KUKA KRL program: MyProgram_211().src

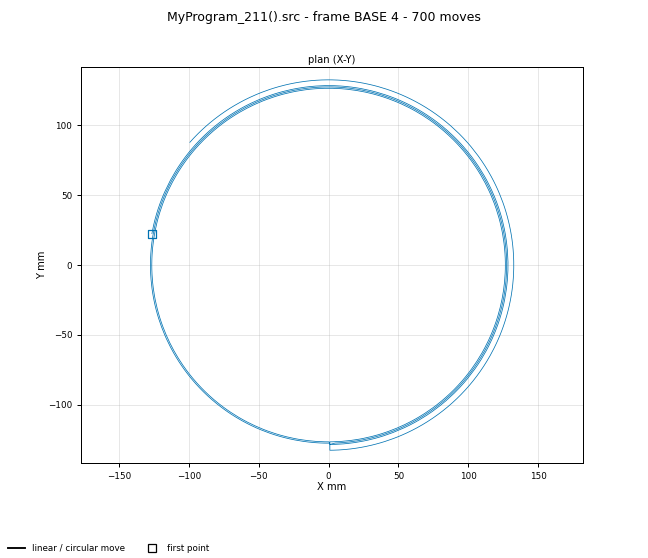
[picture p0: tool path of MyProgram_211().src in frame BASE 4, 700 of 700 moves have a stored position in this frame; points joined in program order, loops and branches not executed]
&ACCESS RVP
&REL 1
&PARAM TEMPLATE = C:\KRC\Roboter\Template\vorgabe
&PARAM EDITMASK = *
DEF MyProgram_211()
; ---- Setting reference (Base) ----
$BASE = BASE_DATA[4]

; --------------------------
; ---- Setting tool (TCP) ----
$TOOL = TOOL_DATA[3]
; --------------------------

$VEL.CP = VEL_APROX_PRINT
Startdeposition()
$VEL.CP = VEL_PRINT
LIN {X -126.5024,Y 22.5306,Z 149,A 167.0251,B 21.3355,C -0.911,E1 21.1965,E2 280.5276} C_DIS
LIN {X -125.8833,Y 25.7659,Z 149,A 165.5743,B 21.3353,C -0.9164,E1 21.1973,E2 281.9739} C_DIS
LIN {X -125.2551,Y 28.6636,Z 149,A 164.2083,B 21.3353,C -0.9188,E1 21.1981,E2 283.3427} C_DIS
LIN {X -124.3308,Y 32.4464,Z 149,A 161.9232,B 21.3358,C -0.9032,E1 21.1998,E2 285.6871} C_DIS
LIN {X -123.1759,Y 36.584,Z 149,A 160.1986,B 21.3353,C -0.9164,E1 21.2011,E2 287.387} C_DIS
LIN {X -122.1569,Y 39.8588,Z 149,A 159.0156,B 21.3346,C -0.9344,E1 21.2021,E2 288.5283} C_DIS
LIN {X -120.7931,Y 43.8121,Z 149,A 156.8151,B 21.3349,C -0.9272,E1 21.2042,E2 290.7636} C_DIS
LIN {X -118.9565,Y 48.5809,Z 149,A 154.7384,B 21.3342,C -0.9418,E1 21.2063,E2 292.8137} C_DIS
LIN {X -117.417,Y 52.1895,Z 149,A 152.9389,B 21.3342,C -0.9451,E1 21.2083,E2 294.616} C_DIS
LIN {X -113.3111,Y 60.5932,Z 149,A 148.9309,B 21.3333,C -0.9635,E1 21.2133,E2 298.5988} C_DIS
LIN {X -109.5371,Y 67.1752,Z 149,A 145.6179,B 21.3328,C -0.9757,E1 21.2179,E2 301.8985} C_DIS
LIN {X -107.9534,Y 69.6925,Z 149,A 143.9828,B 21.3332,C -0.9674,E1 21.2204,E2 303.5666} C_DIS
LIN {X -105.4695,Y 73.3966,Z 149,A 141.5266,B 21.3337,C -0.9547,E1 21.2243,E2 306.0723} C_DIS
LIN {X -102.7831,Y 77.1145,Z 149,A 139.5857,B 21.3333,C -0.9642,E1 21.2275,E2 307.9982} C_DIS
LIN {X -100.3563,Y 80.247,Z 149,A 138.1638,B 21.3325,C -0.9821,E1 21.2299,E2 309.3785} C_DIS
LIN {X -97.498,Y 83.6963,Z 149,A 136.0509,B 21.3325,C -0.9827,E1 21.2338,E2 311.5014} C_DIS
LIN {X -95.072,Y 86.442,Z 149,A 134.5353,B 21.3321,C -0.9913,E1 21.2366,E2 313.0012} C_DIS
LIN {X -92.0357,Y 89.6687,Z 149,A 132.5092,B 21.332,C -0.9941,E1 21.2405,E2 315.0301} C_DIS
LIN {X -88.8889,Y 92.7883,Z 149,A 130.6084,B 21.3316,C -1.0016,E1 21.2443,E2 316.9194} C_DIS
LIN {X -86.2647,Y 95.2328,Z 149,A 129.1349,B 21.3313,C -1.0102,E1 21.2472,E2 318.3764} C_DIS
LIN {X -83.3834,Y 97.7657,Z 149,A 127.3435,B 21.3313,C -1.0108,E1 21.251,E2 320.1746} C_DIS
LIN {X -80.3668,Y 100.2607,Z 149,A 125.424,B 21.3313,C -1.0077,E1 21.2552,E2 322.1114} C_DIS
LIN {X -76.5633,Y 103.194,Z 149,A 123.3887,B 21.331,C -1.0163,E1 21.2597,E2 324.1317} C_DIS
LIN {X -73.2443,Y 105.5755,Z 149,A 121.5811,B 21.3308,C -1.0204,E1 21.2638,E2 325.9353} C_DIS
LIN {X -70.1708,Y 107.6429,Z 149,A 119.8567,B 21.3308,C -1.0206,E1 21.2679,E2 327.6658} C_DIS
LIN {X -66.1096,Y 110.1838,Z 149,A 117.7568,B 21.3305,C -1.0259,E1 21.2728,E2 329.759} C_DIS
LIN {X -62.338,Y 112.3601,Z 149,A 115.4206,B 21.3311,C -1.0136,E1 21.2786,E2 332.1374} C_DIS
LIN {X -59.0857,Y 114.1043,Z 149,A 114.1862,B 21.3302,C -1.0326,E1 21.2816,E2 333.3234} C_DIS
LIN {X -55.8111,Y 115.7399,Z 149,A 112.3225,B 21.3305,C -1.0258,E1 21.2863,E2 335.2114} C_DIS
LIN {X -50.8834,Y 117.9885,Z 149,A 110.1116,B 21.33,C -1.0375,E1 21.2919,E2 337.3965} C_DIS
LIN {X -47.6091,Y 119.3482,Z 149,A 108.3813,B 21.3302,C -1.0336,E1 21.2964,E2 339.1421} C_DIS
LIN {X -43.4647,Y 120.9184,Z 149,A 105.8791,B 21.331,C -1.015,E1 21.3031,E2 341.7016} C_DIS
LIN {X -38.7505,Y 122.5111,Z 149,A 104.4896,B 21.3294,C -1.0509,E1 21.3065,E2 342.9952} C_DIS
LIN {X -36.1903,Y 123.2911,Z 149,A 103.0975,B 21.3297,C -1.0441,E1 21.3103,E2 344.4089} C_DIS
LIN {X -32.8603,Y 124.2204,Z 149,A 101.6079,B 21.3295,C -1.0477,E1 21.3143,E2 345.8911} C_DIS
LIN {X -29.7621,Y 124.9992,Z 149,A 100.1887,B 21.3295,C -1.0493,E1 21.3181,E2 347.3085} C_DIS
LIN {X -26.6465,Y 125.7006,Z 149,A 98.734,B 21.3295,C -1.0492,E1 21.3221,E2 348.7656} C_DIS
LIN {X -22.5065,Y 126.5067,Z 149,A 96.5684,B 21.3299,C -1.039,E1 21.3282,E2 350.9621} C_DIS
LIN {X -17.6004,Y 127.2833,Z 149,A 94.5907,B 21.3294,C -1.05,E1 21.3335,E2 352.9113} C_DIS
LIN {X -13.9215,Y 127.7369,Z 149,A 92.2906,B 21.3306,C -1.0244,E1 21.3401,E2 355.2835} C_DIS
LIN {X -8.9034,Y 128.1852,Z 149,A 90.7884,B 21.3292,C -1.0558,E1 21.3441,E2 356.7} C_DIS
LIN {X -2.7081,Y 128.466,Z 149,A 88.0474,B 21.3291,C -1.0576,E1 21.3517,E2 359.4369} C_DIS
LIN {X 4.2169,Y 128.4248,Z 149,A 84.9282,B 21.3291,C -1.0567,E1 21.3604,E2 362.5581} C_DIS
LIN {X 8.7162,Y 128.1989,Z 149,A 82.8985,B 21.3291,C -1.0558,E1 21.3661,E2 364.5895} C_DIS
LIN {X 12.1904,Y 127.9137,Z 149,A 80.8062,B 21.3302,C -1.0331,E1 21.3721,E2 366.7424} C_DIS
LIN {X 16.289,Y 127.4571,Z 149,A 79.4266,B 21.3293,C -1.0519,E1 21.3757,E2 368.0693} C_DIS
LIN {X 20.9637,Y 126.7716,Z 149,A 77.6065,B 21.3288,C -1.0633,E1 21.3807,E2 369.856} C_DIS
LIN {X 23.6917,Y 126.2908,Z 149,A 76.0677,B 21.3294,C -1.05,E1 21.385,E2 371.4294} C_DIS
LIN {X 27.1575,Y 125.5903,Z 149,A 74.566,B 21.3294,C -1.0524,E1 21.3891,E2 372.9223} C_DIS
LIN {X 30.1689,Y 124.9011,Z 149,A 73.1257,B 21.3294,C -1.0489,E1 21.393,E2 374.3696} C_DIS
LIN {X 33.9154,Y 123.9383,Z 149,A 71.31,B 21.3297,C -1.0439,E1 21.3979,E2 376.1957} C_DIS
LIN {X 37.8426,Y 122.7942,Z 149,A 69.6544,B 21.3294,C -1.0497,E1 21.4023,E2 377.8318} C_DIS
LIN {X 40.6135,Y 121.9055,Z 149,A 68.3282,B 21.3295,C -1.0474,E1 21.4058,E2 379.1614} C_DIS
LIN {X 43.7376,Y 120.82,Z 149,A 66.4377,B 21.3304,C -1.0283,E1 21.4109,E2 381.0995} C_DIS
LIN {X 47.3652,Y 119.4465,Z 149,A 64.6738,B 21.3306,C -1.0251,E1 21.4155,E2 382.8676} C_DIS
LIN {X 50.8844,Y 117.9881,Z 149,A 63.4384,B 21.3298,C -1.0431,E1 21.4186,E2 384.0502} C_DIS
LIN {X 54.0438,Y 116.5747,Z 149,A 61.8787,B 21.3298,C -1.0406,E1 21.4225,E2 385.6122} C_DIS
LIN {X 57.0953,Y 115.1112,Z 149,A 60.3886,B 21.3299,C -1.0395,E1 21.4263,E2 387.1004} C_DIS
LIN {X 59.9976,Y 113.6255,Z 149,A 58.904,B 21.3301,C -1.0362,E1 21.43,E2 388.589} C_DIS
LIN {X 63.8911,Y 111.4849,Z 149,A 56.7721,B 21.3305,C -1.0269,E1 21.4352,E2 390.7389} C_DIS
LIN {X 66.7791,Y 109.7796,Z 149,A 55.4128,B 21.3303,C -1.0305,E1 21.4384,E2 392.0832} C_DIS
LIN {X 70.0603,Y 107.7147,Z 149,A 53.6927,B 21.3304,C -1.0282,E1 21.4425,E2 393.8031} C_DIS
LIN {X 74.7579,Y 104.509,Z 149,A 51.1929,B 21.3306,C -1.0255,E1 21.4482,E2 396.3} C_DIS
LIN {X 77.9903,Y 102.1195,Z 149,A 49.3589,B 21.3308,C -1.0205,E1 21.4523,E2 398.1398} C_DIS
LIN {X 81.4914,Y 99.3483,Z 149,A 47.3921,B 21.3309,C -1.0179,E1 21.4566,E2 400.1051} C_DIS
LIN {X 84.7295,Y 96.6018,Z 149,A 45.5153,B 21.331,C -1.0149,E1 21.4605,E2 401.9811} C_DIS
LIN {X 88.9751,Y 92.7059,Z 149,A 42.9302,B 21.3313,C -1.009,E1 21.4658,E2 404.57} C_DIS
LIN {X 91.0131,Y 90.7057,Z 149,A 41.2496,B 21.3322,C -0.9883,E1 21.4693,E2 406.2985} C_DIS
LIN {X 93.9321,Y 87.6793,Z 149,A 39.8186,B 21.3316,C -1.0037,E1 21.4719,E2 407.6799} C_DIS
LIN {X 96.6382,Y 84.6877,Z 149,A 37.9954,B 21.3318,C -0.9986,E1 21.4753,E2 409.5075} C_DIS
LIN {X 99.4168,Y 81.4076,Z 149,A 36.0873,B 21.332,C -0.9945,E1 21.4787,E2 411.4164} C_DIS
LIN {X 102.2616,Y 77.8046,Z 149,A 34.0421,B 21.3322,C -0.9896,E1 21.4822,E2 413.4633} C_DIS
LIN {X 104.8267,Y 74.3124,Z 149,A 31.6772,B 21.3332,C -0.9656,E1 21.4861,E2 415.8801} C_DIS
LIN {X 107.3529,Y 70.6132,Z 149,A 30.6055,B 21.3316,C -1.0018,E1 21.4877,E2 416.8465} C_DIS
LIN {X 111.3736,Y 64.0852,Z 149,A 26.928,B 21.3326,C -0.9812,E1 21.4931,E2 420.5581} C_DIS
LIN {X 113.0317,Y 61.1133,Z 149,A 25.2168,B 21.3331,C -0.9684,E1 21.4954,E2 422.2937} C_DIS
LIN {X 115.1112,Y 57.0953,Z 149,A 23.2364,B 21.3333,C -0.9645,E1 21.4979,E2 424.2721} C_DIS
LIN {X 116.7392,Y 53.6882,Z 149,A 21.636,B 21.3333,C -0.9635,E1 21.4998,E2 425.8648} C_DIS
LIN {X 118.8712,Y 48.7873,Z 149,A 19.1595,B 21.3338,C -0.9525,E1 21.5025,E2 428.3552} C_DIS
LIN {X 120.5097,Y 44.5879,Z 149,A 17.2936,B 21.3338,C -0.9532,E1 21.5043,E2 430.207} C_DIS
LIN {X 121.7655,Y 41.0342,Z 149,A 15.5898,B 21.334,C -0.9472,E1 21.5059,E2 431.9158} C_DIS
LIN {X 122.8444,Y 37.6788,Z 149,A 14.0311,B 21.3342,C -0.9431,E1 21.5072,E2 433.4751} C_DIS
LIN {X 123.7755,Y 34.4973,Z 149,A 12.6305,B 21.3342,C -0.9421,E1 21.5083,E2 434.8687} C_DIS
LIN {X 124.6792,Y 31.0778,Z 149,A 11.0066,B 21.3345,C -0.9352,E1 21.5094,E2 436.5003} C_DIS
LIN {X 125.8354,Y 26.0013,Z 149,A 8.9227,B 21.3344,C -0.9389,E1 21.5107,E2 438.5598} C_DIS
LIN {X 126.5495,Y 22.2671,Z 149,A 7.0765,B 21.3349,C -0.9268,E1 21.5116,E2 440.4261} C_DIS
LIN {X 127.4203,Y 16.5703,Z 149,A 4.5861,B 21.3351,C -0.9224,E1 21.5126,E2 442.9112} C_DIS
LIN {X 128.0462,Y 10.709,Z 149,A 1.804,B 21.3357,C -0.9071,E1 21.5134,E2 445.7154} C_DIS
LIN {X 128.4745,Y 2.2,Z 149,A -2.7502,B 21.3375,C -0.8609,E1 21.5138,E2 450.3633} C_DIS
LIN {X 128.4331,Y -3.9504,Z 149,A -5.6329,B 21.3381,C -0.8459,E1 21.5136,E2 453.2665} C_DIS
LIN {X 128.0339,Y -10.8549,Z 149,A -7.5384,B 21.3364,C -0.8894,E1 21.5132,E2 455.0399} C_DIS
LIN {X 127.3738,Y -16.9253,Z 149,A -10.2869,B 21.3368,C -0.8795,E1 21.5124,E2 457.796} C_DIS
LIN {X 126.0458,Y -24.9673,Z 149,A -14.0539,B 21.3375,C -0.8619,E1 21.5106,E2 461.5848} C_DIS
LIN {X 125.281,Y -28.5505,Z 149,A -15.5989,B 21.3375,C -0.8608,E1 21.5096,E2 463.122} C_DIS
LIN {X 124.5398,Y -31.6271,Z 149,A -16.9744,B 21.3376,C -0.858,E1 21.5087,E2 464.4957} C_DIS
LIN {X 123.6426,Y -34.9726,Z 149,A -18.5415,B 21.3378,C -0.8521,E1 21.5075,E2 466.0681} C_DIS
LIN {X 122.3986,Y -39.1026,Z 149,A -20.4262,B 21.338,C -0.848,E1 21.506,E2 467.9514} C_DIS
LIN {X 121.3036,Y -42.3787,Z 149,A -21.9571,B 21.3382,C -0.8436,E1 21.5046,E2 469.4838} C_DIS
LIN {X 119.49,Y -47.2557,Z 149,A -24.2295,B 21.3383,C -0.8387,E1 21.5024,E2 471.7545} C_DIS
LIN {X 118.2879,Y -50.1888,Z 149,A -25.632,B 21.3385,C -0.835,E1 21.5009,E2 473.1581} C_DIS
LIN {X 117.1157,Y -52.863,Z 149,A -26.9554,B 21.3387,C -0.8301,E1 21.4994,E2 474.4861} C_DIS
LIN {X 114.5241,Y -58.2632,Z 149,A -29.6054,B 21.3389,C -0.8232,E1 21.4961,E2 477.1381} C_DIS
LIN {X 112.8123,Y -61.5165,Z 149,A -31.3116,B 21.3392,C -0.8154,E1 21.4938,E2 478.8549} C_DIS
LIN {X 109.4302,Y -67.3494,Z 149,A -33.9605,B 21.3389,C -0.8231,E1 21.4902,E2 481.4666} C_DIS
LIN {X 107.0779,Y -71.0307,Z 149,A -36.2183,B 21.3396,C -0.8036,E1 21.4867,E2 483.7642} C_DIS
LIN {X 104.7211,Y -74.4612,Z 149,A -38.0778,B 21.3398,C -0.7984,E1 21.4837,E2 485.6271} C_DIS
LIN {X 99.2501,Y -81.6115,Z 149,A -41.8391,B 21.3398,C -0.7992,E1 21.4773,E2 489.3649} C_DIS
LIN {X 97.2041,Y -84.0375,Z 149,A -44.077,B 21.3412,C -0.7586,E1 21.4731,E2 491.7015} C_DIS
LIN {X 93.7509,Y -87.8736,Z 149,A -46.4121,B 21.3414,C -0.7515,E1 21.4686,E2 494.0441} C_DIS
LIN {X 90,Y -91.7109,Z 149,A -48.0087,B 21.3404,C -0.7814,E1 21.4656,E2 495.551} C_DIS
LIN {X 84.0776,Y -97.1696,Z 149,A -51.4099,B 21.3404,C -0.7816,E1 21.4587,E2 498.9351} C_DIS
LIN {X 80.033,Y -100.5266,Z 149,A -53.9677,B 21.3409,C -0.7669,E1 21.4531,E2 501.5215} C_DIS
LIN {X 74.3559,Y -104.7959,Z 149,A -57.3669,B 21.3415,C -0.7501,E1 21.4454,E2 504.9523} C_DIS
LIN {X 70.2672,Y -107.5803,Z 149,A -59.4392,B 21.3415,C -0.7517,E1 21.4406,E2 507.0118} C_DIS
LIN {X 64.9358,Y -110.879,Z 149,A -62.1325,B 21.3415,C -0.7511,E1 21.4342,E2 509.6966} C_DIS
LIN {X 61.8538,Y -112.6283,Z 149,A -63.6817,B 21.3415,C -0.7498,E1 21.4304,E2 511.2441} C_DIS
LIN {X 57.9866,Y -114.665,Z 149,A -65.6063,B 21.3415,C -0.7477,E1 21.4256,E2 513.168} C_DIS
LIN {X 54.2584,Y -116.4755,Z 149,A -67.4216,B 21.3416,C -0.7463,E1 21.421,E2 514.9816} C_DIS
LIN {X 46.0167,Y -119.9717,Z 149,A -71.304,B 21.3416,C -0.7454,E1 21.4111,E2 518.8555} C_DIS
LIN {X 39.0159,Y -122.4263,Z 149,A -74.6753,B 21.3419,C -0.7385,E1 21.4022,E2 522.2378} C_DIS
LIN {X 35.9952,Y -123.3483,Z 149,A -76.0894,B 21.3419,C -0.7367,E1 21.3983,E2 523.6538} C_DIS
LIN {X 32.7815,Y -124.2414,Z 149,A -77.6265,B 21.3421,C -0.733,E1 21.3942,E2 525.1981} C_DIS
LIN {X 28.0427,Y -125.397,Z 149,A -79.7469,B 21.3421,C -0.7333,E1 21.3884,E2 527.3141} C_DIS
LIN {X 25.0664,Y -126.0256,Z 149,A -81.2666,B 21.3423,C -0.7251,E1 21.3842,E2 528.8541} C_DIS
LIN {X 18.7391,Y -127.1205,Z 149,A -83.9386,B 21.3421,C -0.7313,E1 21.3769,E2 531.5058} C_DIS
LIN {X 13.5131,Y -127.7809,Z 149,A -86.3427,B 21.3422,C -0.7275,E1 21.3702,E2 533.918} C_DIS
LIN {X 10.7784,Y -128.0404,Z 149,A -88.4747,B 21.3435,C -0.6883,E1 21.364,E2 536.1563} C_DIS
LIN {X 4.483,Y -128.4161,Z 149,A -90.14,B 21.342,C -0.7361,E1 21.3597,E2 537.6897} C_DIS
LIN {X 0.927,Y -128.4536,Z 149,A -91.6085,B 21.3418,C -0.7412,E1 21.3557,E2 539.144} C_DIS
Enddeposition()
LIN {X 0.927,Y -128.4536,Z 149,A -91.6085,B 21.3418,C -0.7412,E1 21.3557,E2 539.144} C_DIS
Startdeposition()
$VEL.CP = VEL_PRINT
LIN {X 4.7464,Y -127.4561,Z 149,A -89.2402,B 20.1151,C -0.5881,E1 20.1307,E2 537.0751} C_DIS
LIN {X 10.6568,Y -127.0982,Z 149,A -86.5313,B 20.1151,C -0.5911,E1 20.1383,E2 534.3589} C_DIS
LIN {X 14.5444,Y -126.7134,Z 149,A -84.6534,B 20.1148,C -0.5971,E1 20.1435,E2 532.4654} C_DIS
LIN {X 20.2771,Y -125.9232,Z 149,A -81.9669,B 20.1147,C -0.6023,E1 20.151,E2 529.7668} C_DIS
LIN {X 24.4978,Y -125.1705,Z 149,A -80.3198,B 20.115,C -0.5923,E1 20.1554,E2 528.1511} C_DIS
LIN {X 27.9449,Y -124.4458,Z 149,A -78.843,B 20.115,C -0.5894,E1 20.1594,E2 526.6854} C_DIS
LIN {X 30.1986,Y -123.9177,Z 149,A -77.5315,B 20.1147,C -0.6015,E1 20.1631,E2 525.3411} C_DIS
LIN {X 34.1976,Y -122.8739,Z 149,A -75.854,B 20.1149,C -0.596,E1 20.1675,E2 523.6831} C_DIS
LIN {X 36.6862,Y -122.1557,Z 149,A -74.6923,B 20.1149,C -0.5971,E1 20.1706,E2 522.5205} C_DIS
LIN {X 39.4672,Y -121.2858,Z 149,A -73.0131,B 20.1144,C -0.614,E1 20.1752,E2 520.7964} C_DIS
LIN {X 42.6116,Y -120.2171,Z 149,A -71.9127,B 20.1148,C -0.5995,E1 20.178,E2 519.7408} C_DIS
LIN {X 45.5503,Y -119.1348,Z 149,A -70.4147,B 20.1146,C -0.6051,E1 20.1819,E2 518.2307} C_DIS
LIN {X 48.5804,Y -117.9311,Z 149,A -69.0819,B 20.1147,C -0.6017,E1 20.1854,E2 516.9118} C_DIS
LIN {X 52.8709,Y -116.0715,Z 149,A -66.7448,B 20.1143,C -0.6145,E1 20.1914,E2 514.5447} C_DIS
LIN {X 56.4413,Y -114.3756,Z 149,A -65.1143,B 20.1144,C -0.6112,E1 20.1955,E2 512.9292} C_DIS
LIN {X 59.6772,Y -112.7218,Z 149,A -63.326,B 20.1142,C -0.6204,E1 20.1999,E2 511.1208} C_DIS
LIN {X 62.6986,Y -111.0713,Z 149,A -61.2287,B 20.1134,C -0.6464,E1 20.2052,E2 508.9562} C_DIS
LIN {X 67.3098,Y -108.3387,Z 149,A -59.4808,B 20.1141,C -0.6227,E1 20.2092,E2 507.2838} C_DIS
LIN {X 71.0985,Y -105.8914,Z 149,A -57.6121,B 20.1141,C -0.6199,E1 20.2135,E2 505.4312} C_DIS
LIN {X 73.1065,Y -104.5152,Z 149,A -56.4889,B 20.1141,C -0.6233,E1 20.2161,E2 504.3031} C_DIS
LIN {X 76.7611,Y -101.8608,Z 149,A -54.3562,B 20.1138,C -0.6317,E1 20.2209,E2 502.1555} C_DIS
LIN {X 80.2186,Y -99.161,Z 149,A -52.4189,B 20.1138,C -0.6345,E1 20.2251,E2 500.2196} C_DIS
LIN {X 82.5731,Y -97.2089,Z 149,A -50.8736,B 20.1134,C -0.6448,E1 20.2285,E2 498.6521} C_DIS
LIN {X 87.5263,Y -92.7741,Z 149,A -48.1006,B 20.1135,C -0.6424,E1 20.2342,E2 495.9003} C_DIS
LIN {X 90.4671,Y -89.9088,Z 149,A -46.473,B 20.1137,C -0.6374,E1 20.2374,E2 494.2957} C_DIS
LIN {X 93.8115,Y -86.4135,Z 149,A -43.914,B 20.113,C -0.6592,E1 20.2424,E2 491.6879} C_DIS
LIN {X 97.1984,Y -82.5855,Z 149,A -41.8392,B 20.1131,C -0.6554,E1 20.2461,E2 489.636} C_DIS
LIN {X 99.9768,Y -79.1998,Z 149,A -39.5317,B 20.1125,C -0.6751,E1 20.2502,E2 487.2853} C_DIS
LIN {X 102.1851,Y -76.3291,Z 149,A -38.3444,B 20.113,C -0.6604,E1 20.2521,E2 486.1475} C_DIS
LIN {X 104.4711,Y -73.1699,Z 149,A -36.4435,B 20.1126,C -0.6715,E1 20.2552,E2 484.2264} C_DIS
LIN {X 106.6586,Y -69.9421,Z 149,A -34.6369,B 20.1124,C -0.6787,E1 20.258,E2 482.4106} C_DIS
LIN {X 109.2731,Y -65.7825,Z 149,A -32.7045,B 20.1126,C -0.6729,E1 20.2608,E2 480.5073} C_DIS
LIN {X 111.4856,Y -61.9588,Z 149,A -30.5627,B 20.1122,C -0.6853,E1 20.2638,E2 478.3437} C_DIS
LIN {X 113.45,Y -58.2812,Z 149,A -28.6777,B 20.112,C -0.6912,E1 20.2663,E2 476.4543} C_DIS
LIN {X 115.32,Y -54.4884,Z 149,A -26.8032,B 20.1118,C -0.6957,E1 20.2685,E2 474.5798} C_DIS
LIN {X 116.9069,Y -50.9937,Z 149,A -25.1424,B 20.1118,C -0.698,E1 20.2704,E2 472.9237} C_DIS
LIN {X 118.0942,Y -48.1815,Z 149,A -23.7507,B 20.1116,C -0.703,E1 20.2719,E2 471.5275} C_DIS
LIN {X 119.5931,Y -44.3294,Z 149,A -21.8766,B 20.1114,C -0.7093,E1 20.2738,E2 469.6483} C_DIS
LIN {X 120.9543,Y -40.4662,Z 149,A -20.1202,B 20.1113,C -0.7113,E1 20.2753,E2 467.8988} C_DIS
LIN {X 122.2021,Y -36.5323,Z 149,A -18.2143,B 20.111,C -0.7192,E1 20.2769,E2 465.984} C_DIS
LIN {X 123.1596,Y -33.155,Z 149,A -16.9029,B 20.1112,C -0.7125,E1 20.2779,E2 464.7012} C_DIS
LIN {X 123.8345,Y -30.544,Z 149,A -15.6412,B 20.111,C -0.7184,E1 20.2787,E2 463.4318} C_DIS
LIN {X 124.6724,Y -26.9119,Z 149,A -13.9981,B 20.111,C -0.7223,E1 20.2797,E2 461.7896} C_DIS
LIN {X 125.4148,Y -23.2198,Z 149,A -11.8715,B 20.1101,C -0.7464,E1 20.2809,E2 459.6092} C_DIS
LIN {X 125.9857,Y -19.8801,Z 149,A -10.6929,B 20.1104,C -0.7363,E1 20.2814,E2 458.4687} C_DIS
LIN {X 126.4932,Y -16.3412,Z 149,A -9.1436,B 20.1104,C -0.7389,E1 20.282,E2 456.9234} C_DIS
LIN {X 127.0258,Y -11.508,Z 149,A -6.8324,B 20.1099,C -0.7512,E1 20.2826,E2 454.594} C_DIS
LIN {X 127.4544,Y -4.79,Z 149,A -3.9482,B 20.1098,C -0.7547,E1 20.2831,E2 451.7216} C_DIS
LIN {X 127.5431,Y -0.7829,Z 149,A -2.3585,B 20.1098,C -0.7512,E1 20.2831,E2 450.1539} C_DIS
LIN {X 127.5386,Y 1.3934,Z 149,A -1.0105,B 20.1092,C -0.7703,E1 20.2831,E2 448.761} C_DIS
LIN {X 127.3088,Y 7.7466,Z 149,A 1.6085,B 20.1092,C -0.769,E1 20.2828,E2 446.1655} C_DIS
LIN {X 127.0669,Y 11.0279,Z 149,A 3.4665,B 20.1085,C -0.7901,E1 20.2823,E2 444.2607} C_DIS
LIN {X 126.7039,Y 14.624,Z 149,A 4.5587,B 20.1091,C -0.7721,E1 20.282,E2 443.2286} C_DIS
LIN {X 126.33,Y 17.5632,Z 149,A 6.1961,B 20.1085,C -0.7895,E1 20.2814,E2 441.5534} C_DIS
LIN {X 125.6211,Y 22.0679,Z 149,A 8.124,B 20.1085,C -0.7905,E1 20.2805,E2 439.6367} C_DIS
LIN {X 124.9645,Y 25.5218,Z 149,A 9.662,B 20.1083,C -0.7936,E1 20.2797,E2 438.1014} C_DIS
LIN {X 124.0672,Y 29.5785,Z 149,A 11.5048,B 20.1082,C -0.7982,E1 20.2785,E2 436.2588} C_DIS
LIN {X 123.21,Y 32.9662,Z 149,A 13.0087,B 20.1081,C -0.8001,E1 20.2775,E2 434.7605} C_DIS
LIN {X 122.1896,Y 36.5752,Z 149,A 14.8393,B 20.1077,C -0.8113,E1 20.276,E2 432.9107} C_DIS
LIN {X 121.0359,Y 40.2211,Z 149,A 16.3953,B 20.1077,C -0.8095,E1 20.2747,E2 431.3713} C_DIS
LIN {X 120.0394,Y 43.1044,Z 149,A 17.6722,B 20.1077,C -0.8095,E1 20.2735,E2 430.1036} C_DIS
LIN {X 118.7515,Y 46.5362,Z 149,A 20.0383,B 20.1063,C -0.8451,E1 20.271,E2 427.6511} C_DIS
LIN {X 116.8757,Y 51.0658,Z 149,A 21.6648,B 20.1071,C -0.8265,E1 20.2693,E2 426.0897} C_DIS
LIN {X 115.2402,Y 54.6554,Z 149,A 23.2898,B 20.1071,C -0.8252,E1 20.2674,E2 424.4797} C_DIS
LIN {X 113.8685,Y 57.4592,Z 149,A 24.7854,B 20.1068,C -0.833,E1 20.2655,E2 422.9717} C_DIS
LIN {X 112.2129,Y 60.632,Z 149,A 26.3084,B 20.1068,C -0.8337,E1 20.2635,E2 421.4569} C_DIS
LIN {X 110.4465,Y 63.7925,Z 149,A 28.2286,B 20.1061,C -0.8506,E1 20.2608,E2 419.5005} C_DIS
LIN {X 107.6365,Y 68.4283,Z 149,A 30.4575,B 20.1062,C -0.8481,E1 20.2576,E2 417.2933} C_DIS
LIN {X 105.4984,Y 71.68,Z 149,A 31.9376,B 20.1065,C -0.8411,E1 20.2553,E2 415.8426} C_DIS
LIN {X 103.4808,Y 74.5637,Z 149,A 33.7991,B 20.1058,C -0.8569,E1 20.2523,E2 413.947} C_DIS
LIN {X 100.8277,Y 78.1132,Z 149,A 35.7478,B 20.1058,C -0.8599,E1 20.249,E2 412.0014} C_DIS
LIN {X 98.1571,Y 81.4438,Z 149,A 37.6229,B 20.1056,C -0.8626,E1 20.2457,E2 410.1297} C_DIS
LIN {X 95.3109,Y 84.7577,Z 149,A 39.6077,B 20.1054,C -0.868,E1 20.242,E2 408.1407} C_DIS
LIN {X 92.5118,Y 87.8043,Z 149,A 41.5229,B 20.1051,C -0.8744,E1 20.2384,E2 406.2174} C_DIS
LIN {X 89.8024,Y 90.5728,Z 149,A 43.1133,B 20.1052,C -0.8718,E1 20.2353,E2 404.6431} C_DIS
LIN {X 87.0279,Y 93.2419,Z 149,A 44.9661,B 20.1049,C -0.8805,E1 20.2315,E2 402.7748} C_DIS
LIN {X 83.5186,Y 96.3985,Z 149,A 47.0546,B 20.1047,C -0.8833,E1 20.2271,E2 400.6887} C_DIS
LIN {X 80.1994,Y 99.1765,Z 149,A 48.9437,B 20.1047,C -0.8847,E1 20.223,E2 398.8049} C_DIS
LIN {X 76.7252,Y 101.8879,Z 149,A 50.9032,B 20.1046,C -0.8874,E1 20.2187,E2 396.8467} C_DIS
LIN {X 74.4583,Y 103.5566,Z 149,A 52.1346,B 20.1046,C -0.8882,E1 20.2159,E2 395.6185} C_DIS
LIN {X 71.1523,Y 105.8553,Z 149,A 54.0001,B 20.1043,C -0.8935,E1 20.2116,E2 393.7457} C_DIS
LIN {X 67.5659,Y 108.1794,Z 149,A 55.8938,B 20.1043,C -0.8954,E1 20.2071,E2 391.8542} C_DIS
LIN {X 63.7265,Y 110.4847,Z 149,A 57.9273,B 20.1041,C -0.8992,E1 20.2022,E2 389.8176} C_DIS
LIN {X 59.8971,Y 112.6063,Z 149,A 59.697,B 20.1043,C -0.8938,E1 20.1979,E2 388.07} C_DIS
LIN {X 56.877,Y 114.1606,Z 149,A 61.3001,B 20.1041,C -0.899,E1 20.1939,E2 386.4575} C_DIS
LIN {X 54.2032,Y 115.4555,Z 149,A 62.7031,B 20.1039,C -0.9034,E1 20.1904,E2 385.0464} C_DIS
LIN {X 50.8033,Y 116.9892,Z 149,A 64.2364,B 20.1041,C -0.8995,E1 20.1865,E2 383.5292} C_DIS
LIN {X 47.2121,Y 118.485,Z 149,A 66.0127,B 20.1039,C -0.9025,E1 20.1819,E2 381.7494} C_DIS
LIN {X 44.4748,Y 119.5387,Z 149,A 67.4781,B 20.1036,C -0.9098,E1 20.178,E2 380.2669} C_DIS
LIN {X 40.4823,Y 120.949,Z 149,A 69.1455,B 20.104,C -0.902,E1 20.1737,E2 378.6263} C_DIS
LIN {X 38.0528,Y 121.7374,Z 149,A 70.3513,B 20.1038,C -0.9052,E1 20.1705,E2 377.414} C_DIS
LIN {X 34.4558,Y 122.8017,Z 149,A 72.0961,B 20.1037,C -0.9089,E1 20.1658,E2 375.6623} C_DIS
LIN {X 30.6803,Y 123.801,Z 149,A 73.9331,B 20.1035,C -0.9133,E1 20.1608,E2 373.8161} C_DIS
LIN {X 26.9047,Y 124.674,Z 149,A 75.3977,B 20.1039,C -0.9032,E1 20.1569,E2 372.3833} C_DIS
LIN {X 24.6177,Y 125.1475,Z 149,A 76.773,B 20.1033,C -0.9167,E1 20.153,E2 370.971} C_DIS
LIN {X 20.9027,Y 125.8196,Z 149,A 78.2077,B 20.1037,C -0.9069,E1 20.1491,E2 369.5665} C_DIS
LIN {X 17.4112,Y 126.3517,Z 149,A 79.8377,B 20.1037,C -0.9091,E1 20.1446,E2 367.9321} C_DIS
LIN {X 15.1294,Y 126.6436,Z 149,A 81.0471,B 20.1033,C -0.9164,E1 20.1412,E2 366.7028} C_DIS
LIN {X 11.1743,Y 127.0545,Z 149,A 82.7566,B 20.1035,C -0.9136,E1 20.1365,E2 365.0027} C_DIS
LIN {X 7.1333,Y 127.3466,Z 149,A 84.6529,B 20.1033,C -0.9167,E1 20.1312,E2 363.0984} C_DIS
LIN {X 2.2615,Y 127.5243,Z 149,A 86.9103,B 20.1033,C -0.9192,E1 20.1249,E2 360.8342} C_DIS
LIN {X -2.2666,Y 127.5243,Z 149,A 88.7583,B 20.1035,C -0.9115,E1 20.1198,E2 359.0085} C_DIS
LIN {X -5.2627,Y 127.436,Z 149,A 90.328,B 20.1032,C -0.9199,E1 20.1153,E2 357.4141} C_DIS
LIN {X -9.6481,Y 127.1793,Z 149,A 91.9754,B 20.1038,C -0.9065,E1 20.1108,E2 355.8051} C_DIS
LIN {X -13.4539,Y 126.8327,Z 149,A 93.8232,B 20.1036,C -0.9108,E1 20.1056,E2 353.9435} C_DIS
LIN {X -17.1777,Y 126.3835,Z 149,A 95.5935,B 20.1035,C -0.9132,E1 20.1007,E2 352.1646} C_DIS
LIN {X -20.9353,Y 125.8141,Z 149,A 97.6306,B 20.103,C -0.9249,E1 20.095,E2 350.0909} C_DIS
LIN {X -24.843,Y 125.1026,Z 149,A 99.0109,B 20.1037,C -0.9079,E1 20.0914,E2 348.7583} C_DIS
LIN {X -28.3557,Y 124.352,Z 149,A 100.6302,B 20.1037,C -0.9068,E1 20.0869,E2 347.1395} C_DIS
LIN {X -32.5013,Y 123.3339,Z 149,A 102.5305,B 20.1039,C -0.9044,E1 20.0818,E2 345.2429} C_DIS
LIN {X -35.763,Y 122.4273,Z 149,A 104.0368,B 20.1039,C -0.9023,E1 20.0778,E2 343.7396} C_DIS
LIN {X -38.6,Y 121.5629,Z 149,A 105.5379,B 20.1037,C -0.9073,E1 20.0737,E2 342.2205} C_DIS
LIN {X -42.9566,Y 120.0927,Z 149,A 107.2675,B 20.1044,C -0.8921,E1 20.0693,E2 340.5311} C_DIS
LIN {X -46.0957,Y 118.9227,Z 149,A 108.9684,B 20.1041,C -0.8977,E1 20.0648,E2 338.8094} C_DIS
LIN {X -48.6277,Y 117.9113,Z 149,A 110.075,B 20.1044,C -0.8916,E1 20.0619,E2 337.7176} C_DIS
LIN {X -51.9006,Y 116.5065,Z 149,A 111.5922,B 20.1046,C -0.8862,E1 20.0581,E2 336.2114} C_DIS
LIN {X -54.7685,Y 115.1862,Z 149,A 112.9697,B 20.1048,C -0.8826,E1 20.0546,E2 334.8401} C_DIS
LIN {X -57.5217,Y 113.8367,Z 149,A 114.4127,B 20.1048,C -0.883,E1 20.051,E2 333.3912} C_DIS
LIN {X -59.98,Y 112.5628,Z 149,A 116.2964,B 20.1038,C -0.9052,E1 20.0462,E2 331.436} C_DIS
LIN {X -63.3869,Y 110.6799,Z 149,A 117.6996,B 20.1045,C -0.8891,E1 20.0429,E2 330.0743} C_DIS
LIN {X -66.9065,Y 108.5886,Z 149,A 119.4603,B 20.1048,C -0.883,E1 20.0387,E2 328.3249} C_DIS
LIN {X -69.8276,Y 106.7339,Z 149,A 121.144,B 20.1047,C -0.885,E1 20.0347,E2 326.6283} C_DIS
LIN {X -72.6774,Y 104.8138,Z 149,A 122.7521,B 20.1047,C -0.8845,E1 20.031,E2 325.0148} C_DIS
LIN {X -79.2919,Y 99.9035,Z 149,A 126.3763,B 20.1051,C -0.8741,E1 20.023,E2 321.4043} C_DIS
LIN {X -82.6591,Y 97.1358,Z 149,A 128.1909,B 20.1055,C -0.8646,E1 20.0191,E2 319.6086} C_DIS
LIN {X -85.2323,Y 94.8861,Z 149,A 129.816,B 20.1055,C -0.8646,E1 20.0157,E2 317.9754} C_DIS
LIN {X -87.8539,Y 92.4647,Z 149,A 131.4932,B 20.1055,C -0.8637,E1 20.0123,E2 316.292} C_DIS
LIN {X -90.8692,Y 89.5028,Z 149,A 133.3784,B 20.1058,C -0.8588,E1 20.0085,E2 314.4111} C_DIS
LIN {X -93.7,Y 86.5349,Z 149,A 135.2228,B 20.1059,C -0.8544,E1 20.005,E2 312.569} C_DIS
LIN {X -98.0299,Y 81.5974,Z 149,A 138.2179,B 20.1062,C -0.8488,E1 19.9996,E2 309.5733} C_DIS
LIN {X -100.1839,Y 78.9374,Z 149,A 139.8469,B 20.1062,C -0.8482,E1 19.9967,E2 307.9362} C_DIS
LIN {X -103.0608,Y 75.1431,Z 149,A 141.6947,B 20.1068,C -0.8319,E1 19.9937,E2 306.1247} C_DIS
LIN {X -105.0614,Y 72.3189,Z 149,A 143.5079,B 20.1066,C -0.8373,E1 19.9907,E2 304.2845} C_DIS
LIN {X -107.3934,Y 68.8081,Z 149,A 145.3981,B 20.1068,C -0.832,E1 19.9879,E2 302.3975} C_DIS
LIN {X -110.3728,Y 63.9198,Z 149,A 147.9996,B 20.1071,C -0.826,E1 19.9841,E2 299.7967} C_DIS
LIN {X -112.3678,Y 60.3438,Z 149,A 149.9215,B 20.1071,C -0.8238,E1 19.9816,E2 297.8682} C_DIS
LIN {X -114.1182,Y 56.9632,Z 149,A 151.3879,B 20.1077,C -0.81,E1 19.9797,E2 296.4322} C_DIS
LIN {X -116.4988,Y 51.9178,Z 149,A 154.0187,B 20.1078,C -0.8072,E1 19.9766,E2 293.7912} C_DIS
LIN {X -117.9155,Y 48.6177,Z 149,A 155.7724,B 20.1078,C -0.8075,E1 19.9747,E2 292.0242} C_DIS
LIN {X -119.2491,Y 45.248,Z 149,A 157.709,B 20.1076,C -0.814,E1 19.9728,E2 290.0549} C_DIS
LIN {X -120.5186,Y 41.7456,Z 149,A 159.0346,B 20.1082,C -0.7962,E1 19.9716,E2 288.7717} C_DIS
LIN {X -122.0086,Y 37.1668,Z 149,A 162.0284,B 20.1073,C -0.8201,E1 19.9691,E2 285.686} C_DIS
LIN {X -123.6286,Y 31.3597,Z 149,A 163.9221,B 20.1088,C -0.7819,E1 19.9678,E2 283.8903} C_DIS
LIN {X -124.6183,Y 27.1627,Z 149,A 165.8228,B 20.109,C -0.7745,E1 19.9666,E2 281.9968} C_DIS
LIN {X -125.2882,Y 23.8822,Z 149,A 167.312,B 20.1092,C -0.7693,E1 19.9658,E2 280.5117} C_DIS
LIN {X -125.8115,Y 20.9514,Z 149,A 168.6053,B 20.1095,C -0.7636,E1 19.9652,E2 279.2255} C_DIS
LIN {X -126.206,Y 18.4305,Z 149,A 169.7626,B 20.1095,C -0.7604,E1 19.9647,E2 278.0687} C_DIS
LIN {X -126.5508,Y 15.9014,Z 149,A 171.1301,B 20.1095,C -0.7648,E1 19.9642,E2 276.6779} C_DIS
LIN {X -126.9669,Y 12.1213,Z 149,A 172.7663,B 20.1097,C -0.7568,E1 19.9637,E2 275.0525} C_DIS
LIN {X -127.2828,Y 8.168,Z 149,A 174.3674,B 20.1101,C -0.7447,E1 19.9634,E2 273.4748} C_DIS
LIN {X -127.4555,Y 4.7614,Z 149,A 176.013,B 20.1101,C -0.744,E1 19.9632,E2 271.8186} C_DIS
LIN {X -127.5455,Y 0.4589,Z 149,A 178.0199,B 20.1103,C -0.7405,E1 19.9632,E2 269.8063} C_DIS
LIN {X -127.5128,Y -2.9042,Z 149,A 179.5641,B 20.1103,C -0.737,E1 19.9632,E2 268.2606} C_DIS
LIN {X -127.3753,Y -6.5633,Z 149,A -178.8522,B 20.1107,C -0.7297,E1 19.9634,E2 266.6863} C_DIS
LIN {X -127.1329,Y -10.2465,Z 149,A -177.0899,B 20.1107,C -0.7283,E1 19.9638,E2 264.9145} C_DIS
LIN {X -126.8181,Y -13.5899,Z 149,A -175.7136,B 20.111,C -0.7188,E1 19.9641,E2 263.5555} C_DIS
LIN {X -126.4683,Y -16.5311,Z 149,A -174.2246,B 20.111,C -0.7204,E1 19.9647,E2 262.0503} C_DIS
LIN {X -125.9177,Y -20.315,Z 149,A -172.5667,B 20.1112,C -0.7129,E1 19.9654,E2 260.4018} C_DIS
LIN {X -125.255,Y -24.0558,Z 149,A -170.7899,B 20.1113,C -0.7103,E1 19.9663,E2 258.6193} C_DIS
LIN {X -124.4091,Y -28.1057,Z 149,A -168.9219,B 20.1115,C -0.705,E1 19.9674,E2 256.7528} C_DIS
LIN {X -123.5859,Y -31.5279,Z 149,A -167.3046,B 20.1116,C -0.7016,E1 19.9684,E2 255.1334} C_DIS
LIN {X -122.6146,Y -35.1234,Z 149,A -165.3366,B 20.1114,C -0.7074,E1 19.97,E2 253.1339} C_DIS
LIN {X -121.6874,Y -38.21,Z 149,A -164.2858,B 20.112,C -0.6886,E1 19.9708,E2 252.1305} C_DIS
LIN {X -119.5505,Y -44.4432,Z 149,A -161.4316,B 20.1125,C -0.6761,E1 19.9734,E2 249.2923} C_DIS
LIN {X -118.2842,Y -47.7103,Z 149,A -159.6449,B 20.1123,C -0.6794,E1 19.9752,E2 247.4833} C_DIS
LIN {X -117.1568,Y -50.4158,Z 149,A -158.317,B 20.1125,C -0.6761,E1 19.9767,E2 246.1556} C_DIS
LIN {X -116.0963,Y -52.8172,Z 149,A -156.9727,B 20.1124,C -0.6788,E1 19.9783,E2 244.7938} C_DIS
LIN {X -114.4777,Y -56.2343,Z 149,A -155.4298,B 20.1127,C -0.6684,E1 19.9801,E2 243.2707} C_DIS
LIN {X -113.1428,Y -58.8755,Z 149,A -153.9619,B 20.1127,C -0.6699,E1 19.982,E2 241.7883} C_DIS
LIN {X -110.9964,Y -62.8316,Z 149,A -151.9097,B 20.1127,C -0.6657,E1 19.9848,E2 239.7349} C_DIS
LIN {X -109.137,Y -66.0076,Z 149,A -150.3256,B 20.113,C -0.6588,E1 19.987,E2 238.1605} C_DIS
LIN {X -107.3148,Y -68.9308,Z 149,A -148.8634,B 20.1132,C -0.6517,E1 19.9892,E2 236.7097} C_DIS
LIN {X -105.3297,Y -71.9279,Z 149,A -147.0576,B 20.1132,C -0.6547,E1 19.9921,E2 234.8835} C_DIS
LIN {X -103.1048,Y -75.0824,Z 149,A -145.5418,B 20.1135,C -0.6424,E1 19.9945,E2 233.3945} C_DIS
LIN {X -100.161,Y -78.9666,Z 149,A -143.1601,B 20.1135,C -0.6443,E1 19.9986,E2 230.9926} C_DIS
LIN {X -97.4657,Y -82.2707,Z 149,A -141.186,B 20.1135,C -0.6421,E1 20.0021,E2 229.0134} C_DIS
LIN {X -94.9587,Y -85.1513,Z 149,A -139.4874,B 20.1137,C -0.6377,E1 20.0052,E2 227.3181} C_DIS
LIN {X -92.24,Y -88.089,Z 149,A -137.7299,B 20.1138,C -0.6323,E1 20.0086,E2 225.5667} C_DIS
LIN {X -89.6438,Y -90.7304,Z 149,A -135.9783,B 20.1138,C -0.6321,E1 20.0121,E2 223.8061} C_DIS
LIN {X -86.5684,Y -93.6692,Z 149,A -134.0461,B 20.1139,C -0.6291,E1 20.016,E2 221.8728} C_DIS
LIN {X -83.2012,Y -96.6719,Z 149,A -132.0625,B 20.1141,C -0.6235,E1 20.0202,E2 219.8954} C_DIS
LIN {X -79.7523,Y -99.537,Z 149,A -129.9898,B 20.1141,C -0.622,E1 20.0246,E2 217.8171} C_DIS
LIN {X -75.8513,Y -102.5409,Z 149,A -127.7711,B 20.1142,C -0.6184,E1 20.0296,E2 215.5987} C_DIS
LIN {X -72.7715,Y -104.7483,Z 149,A -126.1242,B 20.1144,C -0.6135,E1 20.0333,E2 213.959} C_DIS
LIN {X -69.7937,Y -106.7562,Z 149,A -124.4495,B 20.1144,C -0.6133,E1 20.0373,E2 212.2779} C_DIS
LIN {X -66.1084,Y -109.076,Z 149,A -122.4994,B 20.1144,C -0.6102,E1 20.0419,E2 210.3293} C_DIS
LIN {X -62.1675,Y -111.3698,Z 149,A -120.4333,B 20.1145,C -0.608,E1 20.0469,E2 208.2617} C_DIS
LIN {X -58.1656,Y -113.5089,Z 149,A -118.5296,B 20.1148,C -0.6002,E1 20.0516,E2 206.3742} C_DIS
LIN {X -55.1655,Y -114.9965,Z 149,A -117.0153,B 20.1148,C -0.5987,E1 20.0554,E2 204.859} C_DIS
LIN {X -51.4228,Y -116.7203,Z 149,A -114.9865,B 20.1147,C -0.6036,E1 20.0606,E2 202.8099} C_DIS
LIN {X -48.4258,Y -117.9957,Z 149,A -113.6893,B 20.1149,C -0.5956,E1 20.0639,E2 201.5323} C_DIS
LIN {X -45.0796,Y -119.3121,Z 149,A -112.0216,B 20.1149,C -0.5961,E1 20.0682,E2 199.8585} C_DIS
LIN {X -42.2323,Y -120.3499,Z 149,A -110.6173,B 20.1149,C -0.5966,E1 20.072,E2 198.4493} C_DIS
LIN {X -38.676,Y -121.5386,Z 149,A -109.0185,B 20.1149,C -0.5919,E1 20.0762,E2 196.8604} C_DIS
LIN {X -35.1256,Y -122.614,Z 149,A -107.2625,B 20.1149,C -0.5942,E1 20.0809,E2 195.094} C_DIS
LIN {X -31.8195,Y -123.5119,Z 149,A -105.6629,B 20.1149,C -0.5957,E1 20.0852,E2 193.4871} C_DIS
LIN {X -27.8396,Y -124.4699,Z 149,A -103.9828,B 20.1151,C -0.5884,E1 20.0898,E2 191.8253} C_DIS
LIN {X -24.2086,Y -125.2258,Z 149,A -102.3434,B 20.1151,C -0.5867,E1 20.0942,E2 190.1888} C_DIS
LIN {X -20.875,Y -125.8242,Z 149,A -100.7751,B 20.1151,C -0.588,E1 20.0986,E2 188.6146} C_DIS
LIN {X -18.3822,Y -126.2129,Z 149,A -99.488,B 20.1149,C -0.5938,E1 20.1022,E2 187.3092} C_DIS
LIN {X -14.3291,Y -126.7385,Z 149,A -97.6212,B 20.1149,C -0.5947,E1 20.1074,E2 185.4383} C_DIS
LIN {X -9.8848,Y -127.162,Z 149,A -95.8739,B 20.1152,C -0.5842,E1 20.1121,E2 183.7205} C_DIS
LIN {X -6.1257,Y -127.3973,Z 149,A -93.6847,B 20.1146,C -0.6043,E1 20.1184,E2 181.4721} C_DIS
LIN {X -2.4448,Y -127.5212,Z 149,A -92.3935,B 20.1151,C -0.5898,E1 20.1219,E2 180.223} C_DIS
LIN {X 0.9077,Y -127.5369,Z 149,A -90.5501,B 20.1147,C -0.6038,E1 20.1272,E2 178.3389} C_DIS
Enddeposition()
LIN {X 0.9077,Y -127.5369,Z 149,A -90.5501,B 20.1147,C -0.6038,E1 20.1272,E2 178.3389} C_DIS
Startdeposition()
$VEL.CP = VEL_PRINT
LIN {X 0.2172,Y -126.596,Z 149,A -91.5737,B 18.8981,C -0.4142,E1 18.9021,E2 179.8083} C_DIS
LIN {X -2.7456,Y -126.5671,Z 149,A -92.9364,B 18.8981,C -0.4132,E1 18.8983,E2 181.1742} C_DIS
LIN {X -6.2389,Y -126.4414,Z 149,A -94.4072,B 18.8981,C -0.4173,E1 18.8943,E2 182.6328} C_DIS
LIN {X -9.3283,Y -126.251,Z 149,A -95.8547,B 18.8981,C -0.4156,E1 18.8902,E2 184.0863} C_DIS
LIN {X -12.1888,Y -126.007,Z 149,A -97.1867,B 18.8981,C -0.4145,E1 18.8865,E2 185.4225} C_DIS
LIN {X -15.267,Y -125.6714,Z 149,A -98.5765,B 18.8981,C -0.4152,E1 18.8826,E2 186.8114} C_DIS
LIN {X -18.3555,Y -125.2581,Z 149,A -99.9635,B 18.8981,C -0.4164,E1 18.8788,E2 188.1961} C_DIS
LIN {X -21.4166,Y -124.7717,Z 149,A -101.4242,B 18.8981,C -0.4147,E1 18.8748,E2 189.6638} C_DIS
LIN {X -24.1271,Y -124.2751,Z 149,A -102.6552,B 18.8981,C -0.4158,E1 18.8714,E2 190.8932} C_DIS
LIN {X -27.7366,Y -123.5199,Z 149,A -104.2168,B 18.898,C -0.4205,E1 18.8672,E2 192.4429} C_DIS
LIN {X -30.0144,Y -122.9859,Z 149,A -105.5152,B 18.8981,C -0.4124,E1 18.8636,E2 193.7687} C_DIS
LIN {X -34.5656,Y -121.7855,Z 149,A -107.6518,B 18.8981,C -0.4136,E1 18.8578,E2 195.9062} C_DIS
LIN {X -38.0161,Y -120.7531,Z 149,A -109.1929,B 18.8981,C -0.418,E1 18.8537,E2 197.4374} C_DIS
LIN {X -41.1809,Y -119.7099,Z 149,A -110.5591,B 18.8979,C -0.4243,E1 18.8501,E2 198.7874} C_DIS
LIN {X -43.663,Y -118.8292,Z 149,A -111.8474,B 18.8979,C -0.4219,E1 18.8467,E2 200.0867} C_DIS
LIN {X -46.8051,Y -117.6258,Z 149,A -113.3535,B 18.8979,C -0.424,E1 18.8428,E2 201.5908} C_DIS
LIN {X -49.8774,Y -116.3556,Z 149,A -114.8655,B 18.8979,C -0.4253,E1 18.8389,E2 203.1035} C_DIS
LIN {X -52.7209,Y -115.0953,Z 149,A -116.2746,B 18.8979,C -0.4268,E1 18.8353,E2 204.5125} C_DIS
LIN {X -55.5266,Y -113.7686,Z 149,A -117.6812,B 18.8978,C -0.4284,E1 18.8318,E2 205.9191} C_DIS
LIN {X -58.0949,Y -112.48,Z 149,A -119.0028,B 18.8978,C -0.4292,E1 18.8285,E2 207.2428} C_DIS
LIN {X -60.8332,Y -111.0229,Z 149,A -120.503,B 18.8978,C -0.4277,E1 18.8248,E2 208.7537} C_DIS
LIN {X -64.5107,Y -108.9275,Z 149,A -122.4693,B 18.8978,C -0.4286,E1 18.82,E2 210.7251} C_DIS
LIN {X -67.7342,Y -106.9524,Z 149,A -124.0009,B 18.8976,C -0.4374,E1 18.8164,E2 212.2358} C_DIS
LIN {X -69.9462,Y -105.5196,Z 149,A -125.3525,B 18.8976,C -0.4337,E1 18.8132,E2 213.6049} C_DIS
LIN {X -72.7042,Y -103.6384,Z 149,A -126.8145,B 18.8976,C -0.4379,E1 18.8099,E2 215.0608} C_DIS
LIN {X -75.405,Y -101.6899,Z 149,A -128.425,B 18.8976,C -0.4368,E1 18.8063,E2 216.6823} C_DIS
LIN {X -79.1129,Y -98.833,Z 149,A -130.5481,B 18.8976,C -0.4404,E1 18.8016,E2 218.8048} C_DIS
LIN {X -82.19,Y -96.2889,Z 149,A -132.3819,B 18.8975,C -0.4429,E1 18.7977,E2 220.6407} C_DIS
LIN {X -85.5064,Y -93.3563,Z 149,A -134.2855,B 18.8973,C -0.4502,E1 18.7937,E2 222.5318} C_DIS
LIN {X -88.3805,Y -90.6406,Z 149,A -136.1853,B 18.8973,C -0.45,E1 18.7899,E2 224.4429} C_DIS
LIN {X -91.2293,Y -87.7728,Z 149,A -138.0397,B 18.8973,C -0.453,E1 18.7863,E2 226.2988} C_DIS
LIN {X -94.3235,Y -84.4379,Z 149,A -140.077,B 18.8971,C -0.4583,E1 18.7824,E2 228.3321} C_DIS
LIN {X -97.2927,Y -80.9996,Z 149,A -142.04,B 18.8969,C -0.4661,E1 18.7789,E2 230.2831} C_DIS
LIN {X -99.7292,Y -77.9799,Z 149,A -143.8381,B 18.8969,C -0.4687,E1 18.7758,E2 232.0845} C_DIS
LIN {X -101.8116,Y -75.2412,Z 149,A -145.5077,B 18.8969,C -0.4686,E1 18.773,E2 233.7655} C_DIS
LIN {X -104.3963,Y -71.6108,Z 149,A -147.3223,B 18.8966,C -0.4804,E1 18.7701,E2 235.5554} C_DIS
LIN {X -106.1194,Y -69.0317,Z 149,A -148.7907,B 18.8966,C -0.4817,E1 18.7678,E2 237.0298} C_DIS
LIN {X -107.6594,Y -66.6053,Z 149,A -150.1014,B 18.8965,C -0.4847,E1 18.7659,E2 238.3404} C_DIS
LIN {X -109.2583,Y -63.9482,Z 149,A -151.5195,B 18.8964,C -0.4878,E1 18.7639,E2 239.7588} C_DIS
LIN {X -110.7917,Y -61.2529,Z 149,A -152.9708,B 18.8964,C -0.4899,E1 18.7619,E2 241.2141} C_DIS
LIN {X -112.365,Y -58.3154,Z 149,A -154.4582,B 18.8962,C -0.4946,E1 18.7599,E2 242.6975} C_DIS
LIN {X -113.6083,Y -55.8516,Z 149,A -155.732,B 18.8962,C -0.4972,E1 18.7584,E2 243.9726} C_DIS
LIN {X -115.0022,Y -52.9223,Z 149,A -157.1896,B 18.896,C -0.5015,E1 18.7566,E2 245.4275} C_DIS
LIN {X -116.2649,Y -50.0872,Z 149,A -158.6047,B 18.896,C -0.5051,E1 18.755,E2 246.8422} C_DIS
LIN {X -117.5434,Y -47.0096,Z 149,A -160.1263,B 18.8959,C -0.5089,E1 18.7534,E2 248.3636} C_DIS
LIN {X -118.6626,Y -44.1081,Z 149,A -161.5493,B 18.8958,C -0.5124,E1 18.752,E2 249.7867} C_DIS
LIN {X -119.7188,Y -41.1554,Z 149,A -162.9402,B 18.8956,C -0.5174,E1 18.7507,E2 251.1727} C_DIS
LIN {X -120.8299,Y -37.7753,Z 149,A -164.7788,B 18.8957,C -0.5144,E1 18.7492,E2 253.035} C_DIS
LIN {X -121.9483,Y -33.9836,Z 149,A -166.4002,B 18.8954,C -0.5253,E1 18.7479,E2 254.6353} C_DIS
LIN {X -122.7448,Y -30.984,Z 149,A -167.8466,B 18.8954,C -0.5281,E1 18.7469,E2 256.0845} C_DIS
LIN {X -123.5186,Y -27.7426,Z 149,A -169.2713,B 18.8952,C -0.5353,E1 18.746,E2 257.498} C_DIS
LIN {X -124.0778,Y -25.1198,Z 149,A -170.6146,B 18.8952,C -0.5347,E1 18.7452,E2 258.8542} C_DIS
LIN {X -124.693,Y -21.8666,Z 149,A -172.0804,B 18.895,C -0.5403,E1 18.7445,E2 260.3144} C_DIS
LIN {X -125.226,Y -18.5801,Z 149,A -173.6067,B 18.895,C -0.5442,E1 18.7439,E2 261.8409} C_DIS
LIN {X -125.5782,Y -16.0189,Z 149,A -174.8814,B 18.895,C -0.5443,E1 18.7434,E2 263.1256} C_DIS
LIN {X -125.9638,Y -12.6385,Z 149,A -176.4036,B 18.8948,C -0.5496,E1 18.7429,E2 264.6438} C_DIS
LIN {X -126.2357,Y -9.538,Z 149,A -177.7543,B 18.8946,C -0.5559,E1 18.7426,E2 265.986} C_DIS
LIN {X -126.4104,Y -6.8552,Z 149,A -179.0849,B 18.8946,C -0.5559,E1 18.7424,E2 267.3276} C_DIS
LIN {X -126.5576,Y -3.1133,Z 149,A 179.3341,B 18.8943,C -0.5649,E1 18.7423,E2 268.8936} C_DIS
LIN {X -126.5992,Y -0.0168,Z 149,A 177.8753,B 18.8943,C -0.5673,E1 18.7423,E2 270.3568} C_DIS
LIN {X -126.5186,Y 4.4316,Z 149,A 175.7969,B 18.8941,C -0.5714,E1 18.7423,E2 272.4394} C_DIS
LIN {X -126.3713,Y 7.5304,Z 149,A 174.3276,B 18.8941,C -0.5737,E1 18.7426,E2 273.9139} C_DIS
LIN {X -126.0079,Y 12.1798,Z 149,A 172.2964,B 18.8938,C -0.5828,E1 18.7431,E2 275.9332} C_DIS
LIN {X -125.6707,Y 15.2734,Z 149,A 170.8894,B 18.8937,C -0.5873,E1 18.7436,E2 277.3379} C_DIS
LIN {X -125.259,Y 18.3488,Z 149,A 169.4971,B 18.8935,C -0.592,E1 18.7441,E2 278.7268} C_DIS
LIN {X -124.7723,Y 21.4126,Z 149,A 168.029,B 18.8935,C -0.5942,E1 18.7448,E2 280.2} C_DIS
LIN {X -124.2115,Y 24.4599,Z 149,A 166.6658,B 18.8933,C -0.5998,E1 18.7455,E2 281.5567} C_DIS
LIN {X -123.5198,Y 27.7372,Z 149,A 165.2562,B 18.893,C -0.608,E1 18.7463,E2 282.9521} C_DIS
LIN {X -122.8573,Y 30.5406,Z 149,A 163.7279,B 18.8931,C -0.6045,E1 18.7473,E2 284.5035} C_DIS
LIN {X -122.0023,Y 33.7904,Z 149,A 162.1318,B 18.8931,C -0.6067,E1 18.7485,E2 286.1056} C_DIS
LIN {X -120.7505,Y 38.0243,Z 149,A 160.1976,B 18.8928,C -0.6148,E1 18.75,E2 288.0297} C_DIS
LIN {X -119.7108,Y 41.1783,Z 149,A 158.8292,B 18.8925,C -0.6237,E1 18.7512,E2 289.3809} C_DIS
LIN {X -118.7504,Y 43.8737,Z 149,A 157.4346,B 18.8925,C -0.6243,E1 18.7526,E2 290.7846} C_DIS
LIN {X -117.6282,Y 46.7992,Z 149,A 155.888,B 18.8925,C -0.6242,E1 18.7542,E2 292.3433} C_DIS
LIN {X -116.0272,Y 50.6369,Z 149,A 153.9611,B 18.8925,C -0.6282,E1 18.7563,E2 294.2723} C_DIS
LIN {X -114.4315,Y 54.1467,Z 149,A 152.3632,B 18.8921,C -0.6381,E1 18.7581,E2 295.8513} C_DIS
LIN {X -113.073,Y 56.9299,Z 149,A 151.0307,B 18.8919,C -0.6444,E1 18.7598,E2 297.174} C_DIS
LIN {X -111.7539,Y 59.4791,Z 149,A 149.6576,B 18.8919,C -0.6456,E1 18.7616,E2 298.5534} C_DIS
LIN {X -110.1548,Y 62.3921,Z 149,A 148.1168,B 18.8917,C -0.6485,E1 18.7637,E2 300.0961} C_DIS
LIN {X -108.5963,Y 65.0664,Z 149,A 146.7367,B 18.8916,C -0.653,E1 18.7656,E2 301.4717} C_DIS
LIN {X -106.9572,Y 67.7265,Z 149,A 145.2799,B 18.8916,C -0.6554,E1 18.7678,E2 302.9312} C_DIS
LIN {X -104.9313,Y 70.8248,Z 149,A 143.4454,B 18.8916,C -0.6546,E1 18.7706,E2 304.7809} C_DIS
LIN {X -102.5959,Y 74.1674,Z 149,A 141.7406,B 18.8912,C -0.6641,E1 18.7734,E2 306.4675} C_DIS
LIN {X -100.7519,Y 76.6541,Z 149,A 140.1674,B 18.8912,C -0.6619,E1 18.776,E2 308.0577} C_DIS
LIN {X -97.932,Y 80.2249,Z 149,A 138.2007,B 18.891,C -0.6702,E1 18.7794,E2 310.0112} C_DIS
LIN {X -95.299,Y 83.3356,Z 149,A 136.2684,B 18.891,C -0.6718,E1 18.783,E2 311.9506} C_DIS
LIN {X -92.7568,Y 86.1562,Z 149,A 134.5052,B 18.8909,C -0.6744,E1 18.7863,E2 313.7164} C_DIS
LIN {X -89.5163,Y 89.5193,Z 149,A 132.3691,B 18.8907,C -0.6785,E1 18.7905,E2 315.8521} C_DIS
LIN {X -86.1658,Y 92.7479,Z 149,A 130.2678,B 18.8906,C -0.6834,E1 18.7947,E2 317.95} C_DIS
LIN {X -82.7704,Y 95.7904,Z 149,A 128.3161,B 18.8903,C -0.6916,E1 18.7988,E2 319.8867} C_DIS
LIN {X -79.7094,Y 98.3524,Z 149,A 126.5149,B 18.8901,C -0.6955,E1 18.8027,E2 321.685} C_DIS
LIN {X -76.7236,Y 100.6987,Z 149,A 124.6352,B 18.8901,C -0.6935,E1 18.8068,E2 323.5804} C_DIS
LIN {X -73.0914,Y 103.3652,Z 149,A 122.6919,B 18.8899,C -0.7007,E1 18.8112,E2 325.5105} C_DIS
LIN {X -70.5239,Y 105.134,Z 149,A 121.1774,B 18.8899,C -0.6998,E1 18.8147,E2 327.0347} C_DIS
LIN {X -66.5974,Y 107.6643,Z 149,A 119.1967,B 18.8897,C -0.7081,E1 18.8194,E2 328.9982} C_DIS
LIN {X -63.9429,Y 109.2614,Z 149,A 117.7904,B 18.8896,C -0.7104,E1 18.8227,E2 330.4033} C_DIS
LIN {X -60.9086,Y 110.9818,Z 149,A 116.3141,B 18.8894,C -0.7165,E1 18.8263,E2 331.8665} C_DIS
LIN {X -58.262,Y 112.393,Z 149,A 114.8394,B 18.8894,C -0.7146,E1 18.83,E2 333.3527} C_DIS
LIN {X -55.7184,Y 113.674,Z 149,A 113.5459,B 18.8894,C -0.7164,E1 18.8332,E2 334.6453} C_DIS
LIN {X -52.9157,Y 115.0052,Z 149,A 112.1376,B 18.8894,C -0.7182,E1 18.8368,E2 336.0526} C_DIS
LIN {X -50.0825,Y 116.2669,Z 149,A 110.7293,B 18.8892,C -0.72,E1 18.8404,E2 337.4599} C_DIS
LIN {X -47.4531,Y 117.3646,Z 149,A 109.3468,B 18.8893,C -0.7185,E1 18.844,E2 338.8515} C_DIS
LIN {X -44.1123,Y 118.661,Z 149,A 107.8077,B 18.8891,C -0.7233,E1 18.8479,E2 340.3799} C_DIS
LIN {X -41.1913,Y 119.7063,Z 149,A 106.4344,B 18.8891,C -0.726,E1 18.8516,E2 341.7484} C_DIS
LIN {X -38.6712,Y 120.5438,Z 149,A 105.1076,B 18.8891,C -0.723,E1 18.8551,E2 343.0879} C_DIS
LIN {X -35.7639,Y 121.4382,Z 149,A 103.7481,B 18.8891,C -0.725,E1 18.8587,E2 344.4444} C_DIS
LIN {X -32.4771,Y 122.3582,Z 149,A 102.266,B 18.8889,C -0.7286,E1 18.8627,E2 345.9182} C_DIS
LIN {X -29.2469,Y 123.1709,Z 149,A 100.758,B 18.8889,C -0.7299,E1 18.8668,E2 347.4251} C_DIS
LIN {X -26.4442,Y 123.8025,Z 149,A 99.43,B 18.8889,C -0.7299,E1 18.8704,E2 348.7551} C_DIS
LIN {X -23.1507,Y 124.4618,Z 149,A 97.9452,B 18.8888,C -0.7323,E1 18.8745,E2 350.2348} C_DIS
LIN {X -20.0942,Y 124.9922,Z 149,A 96.5086,B 18.8888,C -0.7321,E1 18.8784,E2 351.6741} C_DIS
LIN {X -17.0303,Y 125.4457,Z 149,A 95.0395,B 18.8888,C -0.7305,E1 18.8825,E2 353.1497} C_DIS
LIN {X -12.9863,Y 125.9285,Z 149,A 93.1248,B 18.8889,C -0.7288,E1 18.8879,E2 355.0712} C_DIS
LIN {X -9.5351,Y 126.2359,Z 149,A 91.822,B 18.8885,C -0.7389,E1 18.8914,E2 356.3434} C_DIS
LIN {X -6.1993,Y 126.4434,Z 149,A 90.2303,B 18.8886,C -0.7366,E1 18.8959,E2 357.9432} C_DIS
LIN {X -3.1011,Y 126.5579,Z 149,A 88.8008,B 18.8886,C -0.7359,E1 18.8999,E2 359.3748} C_DIS
LIN {X -0.2303,Y 126.5959,Z 149,A 87.4356,B 18.8887,C -0.7338,E1 18.9037,E2 360.7467} C_DIS
LIN {X 2.9039,Y 126.5634,Z 149,A 86.0443,B 18.8887,C -0.7349,E1 18.9076,E2 362.1344} C_DIS
LIN {X 6.2235,Y 126.4422,Z 149,A 84.6119,B 18.8886,C -0.7375,E1 18.9115,E2 363.5582} C_DIS
LIN {X 9.1323,Y 126.2654,Z 149,A 83.1932,B 18.8887,C -0.7337,E1 18.9155,E2 364.9874} C_DIS
LIN {X 13.2109,Y 125.9043,Z 149,A 81.2782,B 18.8888,C -0.7312,E1 18.9209,E2 366.9087} C_DIS
LIN {X 17.0392,Y 125.4445,Z 149,A 79.6669,B 18.8887,C -0.7356,E1 18.9253,E2 368.5046} C_DIS
LIN {X 19.892,Y 125.0235,Z 149,A 78.3507,B 18.8887,C -0.7348,E1 18.9289,E2 369.8217} C_DIS
LIN {X 23.1737,Y 124.4574,Z 149,A 76.9037,B 18.8887,C -0.7364,E1 18.9329,E2 371.2616} C_DIS
LIN {X 25.9928,Y 123.9,Z 149,A 75.5513,B 18.8887,C -0.7338,E1 18.9366,E2 372.6196} C_DIS
LIN {X 29.0342,Y 123.2222,Z 149,A 74.1223,B 18.8887,C -0.7323,E1 18.9405,E2 374.0504} C_DIS
LIN {X 31.4878,Y 122.6169,Z 149,A 72.8212,B 18.889,C -0.7258,E1 18.9441,E2 375.369} C_DIS
LIN {X 35.2604,Y 121.5856,Z 149,A 71.219,B 18.8888,C -0.7308,E1 18.9483,E2 376.9523} C_DIS
LIN {X 38.4482,Y 120.615,Z 149,A 69.5988,B 18.889,C -0.7254,E1 18.9527,E2 378.5849} C_DIS
LIN {X 42.4241,Y 119.2759,Z 149,A 67.814,B 18.889,C -0.728,E1 18.9573,E2 380.357} C_DIS
LIN {X 45.3536,Y 118.193,Z 149,A 66.415,B 18.889,C -0.7271,E1 18.961,E2 381.7545} C_DIS
LIN {X 48.23,Y 117.0489,Z 149,A 64.885,B 18.8892,C -0.7209,E1 18.965,E2 383.299} C_DIS
LIN {X 52.1146,Y 115.3711,Z 149,A 62.9726,B 18.8892,C -0.7188,E1 18.9699,E2 385.2114} C_DIS
LIN {X 55.523,Y 113.7703,Z 149,A 61.5027,B 18.889,C -0.7256,E1 18.9735,E2 386.6553} C_DIS
LIN {X 58.101,Y 112.4768,Z 149,A 60.1007,B 18.8892,C -0.7202,E1 18.977,E2 388.0685} C_DIS
LIN {X 62.4137,Y 110.1425,Z 149,A 57.8968,B 18.8893,C -0.7178,E1 18.9824,E2 390.2712} C_DIS
LIN {X 65.091,Y 108.5816,Z 149,A 56.4929,B 18.8894,C -0.7157,E1 18.9858,E2 391.6757} C_DIS
LIN {X 67.5236,Y 107.0853,Z 149,A 55.2086,B 18.8894,C -0.714,E1 18.9888,E2 392.9594} C_DIS
LIN {X 70.1381,Y 105.3915,Z 149,A 53.7568,B 18.8896,C -0.7102,E1 18.9922,E2 394.4166} C_DIS
LIN {X 72.6964,Y 103.6438,Z 149,A 52.3041,B 18.8898,C -0.7059,E1 18.9956,E2 395.8755} C_DIS
LIN {X 75.9859,Y 101.2569,Z 149,A 50.4297,B 18.8899,C -0.7014,E1 18.9998,E2 397.7547} C_DIS
LIN {X 79.1996,Y 98.7636,Z 149,A 48.5902,B 18.89,C -0.6981,E1 19.0038,E2 399.595} C_DIS
LIN {X 82.7761,Y 95.7855,Z 149,A 46.5149,B 18.8901,C -0.6953,E1 19.0083,E2 401.668} C_DIS
LIN {X 86.0861,Y 92.8221,Z 149,A 44.5042,B 18.8903,C -0.6913,E1 19.0124,E2 403.6798} C_DIS
LIN {X 89.5168,Y 89.5187,Z 149,A 42.3818,B 18.8903,C -0.6881,E1 19.0166,E2 405.8} C_DIS
LIN {X 92.1464,Y 86.8086,Z 149,A 40.7755,B 18.8903,C -0.6884,E1 19.0197,E2 407.3958} C_DIS
LIN {X 94.8387,Y 83.8589,Z 149,A 38.8863,B 18.8906,C -0.6813,E1 19.0233,E2 409.2956} C_DIS
LIN {X 97.3634,Y 80.9143,Z 149,A 37.1193,B 18.8908,C -0.6768,E1 19.0265,E2 411.0652} C_DIS
LIN {X 100.2716,Y 77.2814,Z 149,A 35.0808,B 18.8908,C -0.6745,E1 19.03,E2 413.0979} C_DIS
LIN {X 102.6146,Y 74.1416,Z 149,A 33.2813,B 18.891,C -0.6692,E1 19.0329,E2 414.9019} C_DIS
LIN {X 105.1396,Y 70.5155,Z 149,A 31.3776,B 18.891,C -0.668,E1 19.0359,E2 416.7965} C_DIS
LIN {X 106.9242,Y 67.7789,Z 149,A 29.9509,B 18.8911,C -0.6663,E1 19.0381,E2 418.2187} C_DIS
LIN {X 108.9448,Y 64.4816,Z 149,A 28.0858,B 18.8914,C -0.6572,E1 19.0408,E2 420.0985} C_DIS
LIN {X 110.7958,Y 61.2454,Z 149,A 26.5091,B 18.8914,C -0.6572,E1 19.0429,E2 421.6644} C_DIS
LIN {X 112.184,Y 58.66,Z 149,A 25.1776,B 18.8916,C -0.6535,E1 19.0447,E2 422.9976} C_DIS
LIN {X 113.6708,Y 55.7248,Z 149,A 23.7489,B 18.8916,C -0.6518,E1 19.0464,E2 424.421} C_DIS
LIN {X 115.0016,Y 52.9235,Z 149,A 22.3574,B 18.8917,C -0.6484,E1 19.0481,E2 425.8127} C_DIS
LIN {X 116.1482,Y 50.3571,Z 149,A 21.0334,B 18.8919,C -0.6428,E1 19.0496,E2 427.1441} C_DIS
LIN {X 117.5473,Y 46.9999,Z 149,A 19.5604,B 18.8919,C -0.645,E1 19.0511,E2 428.5992} C_DIS
LIN {X 118.6275,Y 44.2019,Z 149,A 18.1017,B 18.8921,C -0.6371,E1 19.0526,E2 430.0711} C_DIS
LIN {X 119.9814,Y 40.3842,Z 149,A 16.2293,B 18.8923,C -0.6303,E1 19.0543,E2 431.95} C_DIS
LIN {X 121.1443,Y 36.7478,Z 149,A 14.6157,B 18.8923,C -0.6298,E1 19.0557,E2 433.5527} C_DIS
LIN {X 121.9475,Y 33.9866,Z 149,A 13.2929,B 18.8925,C -0.6251,E1 19.0567,E2 434.8796} C_DIS
LIN {X 122.744,Y 30.9871,Z 149,A 11.8699,B 18.8927,C -0.6202,E1 19.0577,E2 436.3065} C_DIS
LIN {X 123.522,Y 27.7277,Z 149,A 10.4197,B 18.8927,C -0.6183,E1 19.0586,E2 437.7511} C_DIS
LIN {X 124.1646,Y 24.693,Z 149,A 9.0109,B 18.8929,C -0.6139,E1 19.0594,E2 439.1624} C_DIS
LIN {X 124.6926,Y 21.8686,Z 149,A 7.7059,B 18.8929,C -0.6098,E1 19.06,E2 440.4696} C_DIS
LIN {X 125.2257,Y 18.5822,Z 149,A 6.2017,B 18.8931,C -0.6053,E1 19.0607,E2 441.9755} C_DIS
LIN {X 125.617,Y 15.723,Z 149,A 4.8378,B 18.8933,C -0.5989,E1 19.0612,E2 443.3478} C_DIS
LIN {X 125.9872,Y 12.3954,Z 149,A 3.2639,B 18.8935,C -0.592,E1 19.0616,E2 444.9305} C_DIS
LIN {X 126.3096,Y 8.5268,Z 149,A 1.4867,B 18.8937,C -0.5857,E1 19.062,E2 446.7125} C_DIS
LIN {X 126.5021,Y 4.854,Z 149,A 0.0048,B 18.8937,C -0.5879,E1 19.0622,E2 448.1758} C_DIS
LIN {X 126.5873,Y 1.531,Z 149,A -1.3753,B 18.8937,C -0.5881,E1 19.0622,E2 449.5439} C_DIS
LIN {X 126.564,Y -2.8829,Z 149,A -3.4624,B 18.8939,C -0.5784,E1 19.0622,E2 451.6441} C_DIS
LIN {X 126.467,Y -5.73,Z 149,A -4.8136,B 18.8941,C -0.5719,E1 19.062,E2 453.0043} C_DIS
LIN {X 126.2519,Y -9.3172,Z 149,A -6.3304,B 18.8941,C -0.5712,E1 19.0618,E2 454.5109} C_DIS
LIN {X 126.0083,Y -12.1755,Z 149,A -7.653,B 18.8943,C -0.5662,E1 19.0614,E2 455.8381} C_DIS
LIN {X 125.6703,Y -15.2766,Z 149,A -8.9839,B 18.8943,C -0.565,E1 19.061,E2 457.1619} C_DIS
LIN {X 125.2594,Y -18.3464,Z 149,A -10.4028,B 18.8945,C -0.56,E1 19.0604,E2 458.5848} C_DIS
LIN {X 124.7739,Y -21.4036,Z 149,A -11.8498,B 18.8946,C -0.5538,E1 19.0598,E2 460.0392} C_DIS
LIN {X 124.2072,Y -24.4824,Z 149,A -13.2053,B 18.8946,C -0.5519,E1 19.0591,E2 461.3899} C_DIS
LIN {X 123.5193,Y -27.7394,Z 149,A -14.5734,B 18.8946,C -0.5528,E1 19.0583,E2 462.7443} C_DIS
LIN {X 122.8583,Y -30.5366,Z 149,A -16.0646,B 18.895,C -0.5412,E1 19.0573,E2 464.2594} C_DIS
LIN {X 122.011,Y -33.7594,Z 149,A -17.4869,B 18.895,C -0.5401,E1 19.0563,E2 465.674} C_DIS
LIN {X 121.1473,Y -36.7381,Z 149,A -18.8013,B 18.895,C -0.5394,E1 19.0552,E2 466.9803} C_DIS
LIN {X 119.9962,Y -40.3396,Z 149,A -20.7004,B 18.8954,C -0.5267,E1 19.0536,E2 468.9036} C_DIS
LIN {X 118.8405,Y -43.6315,Z 149,A -22.2271,B 18.8954,C -0.5241,E1 19.0521,E2 470.4268} C_DIS
LIN {X 117.6266,Y -46.8031,Z 149,A -23.787,B 18.8956,C -0.5186,E1 19.0505,E2 471.9916} C_DIS
LIN {X 116.006,Y -50.6858,Z 149,A -25.6914,B 18.8958,C -0.5131,E1 19.0484,E2 473.899} C_DIS
LIN {X 114.4443,Y -54.12,Z 149,A -27.2417,B 18.8958,C -0.5144,E1 19.0466,E2 475.4338} C_DIS
LIN {X 113.0851,Y -56.9062,Z 149,A -28.5652,B 18.8958,C -0.5135,E1 19.045,E2 476.7503} C_DIS
LIN {X 111.7595,Y -59.4685,Z 149,A -29.9408,B 18.8959,C -0.507,E1 19.0432,E2 478.1359} C_DIS
LIN {X 109.7651,Y -63.0752,Z 149,A -31.9493,B 18.8962,C -0.4961,E1 19.0404,E2 480.1637} C_DIS
LIN {X 107.7782,Y -66.4125,Z 149,A -33.5339,B 18.8962,C -0.4982,E1 19.0382,E2 481.731} C_DIS
LIN {X 106.2473,Y -68.8348,Z 149,A -34.8195,B 18.8962,C -0.4951,E1 19.0362,E2 483.0172} C_DIS
LIN {X 104.3898,Y -71.6204,Z 149,A -36.2606,B 18.8962,C -0.494,E1 19.034,E2 484.4519} C_DIS
LIN {X 102.6034,Y -74.1571,Z 149,A -37.7112,B 18.8964,C -0.4885,E1 19.0316,E2 485.9099} C_DIS
LIN {X 101.1228,Y -76.1635,Z 149,A -38.9525,B 18.8966,C -0.4811,E1 19.0295,E2 487.1659} C_DIS
LIN {X 98.3466,Y -79.7166,Z 149,A -41.0243,B 18.8967,C -0.4746,E1 19.0259,E2 489.2442} C_DIS
LIN {X 95.7872,Y -82.7741,Z 149,A -42.7923,B 18.8967,C -0.4716,E1 19.0227,E2 491.0105} C_DIS
LIN {X 92.806,Y -86.1034,Z 149,A -44.6871,B 18.8967,C -0.4718,E1 19.0192,E2 492.8934} C_DIS
LIN {X 90.0551,Y -88.9769,Z 149,A -46.61,B 18.897,C -0.4627,E1 19.0154,E2 494.8329} C_DIS
LIN {X 86.8157,Y -92.1397,Z 149,A -48.5157,B 18.897,C -0.4636,E1 19.0116,E2 496.7249} C_DIS
LIN {X 83.923,Y -94.7821,Z 149,A -50.4036,B 18.8972,C -0.4552,E1 19.0076,E2 498.6284} C_DIS
LIN {X 80.8129,Y -97.4473,Z 149,A -52.2179,B 18.8972,C -0.4528,E1 19.0038,E2 500.4406} C_DIS
LIN {X 77.2746,Y -100.2769,Z 149,A -54.2553,B 18.8973,C -0.4491,E1 18.9993,E2 502.479} C_DIS
LIN {X 74.3589,Y -102.4571,Z 149,A -55.7783,B 18.8973,C -0.4507,E1 18.9959,E2 503.9898} C_DIS
LIN {X 71.612,Y -104.3955,Z 149,A -57.229,B 18.8973,C -0.4505,E1 18.9926,E2 505.4342} C_DIS
LIN {X 69.0333,Y -106.1184,Z 149,A -58.819,B 18.8975,C -0.4406,E1 18.9888,E2 507.0473} C_DIS
LIN {X 65.2349,Y -108.4952,Z 149,A -60.7025,B 18.8975,C -0.4426,E1 18.9844,E2 508.9166} C_DIS
LIN {X 62.5889,Y -110.0425,Z 149,A -62.0804,B 18.8975,C -0.4406,E1 18.981,E2 510.295} C_DIS
LIN {X 59.6994,Y -111.6367,Z 149,A -63.5954,B 18.8975,C -0.4373,E1 18.9773,E2 511.8143} C_DIS
LIN {X 56.9189,Y -113.0786,Z 149,A -64.9326,B 18.8975,C -0.4382,E1 18.974,E2 513.1437} C_DIS
LIN {X 54.3276,Y -114.3451,Z 149,A -66.2816,B 18.8976,C -0.4346,E1 18.9706,E2 514.4991} C_DIS
LIN {X 51.4869,Y -115.6519,Z 149,A -67.6897,B 18.8976,C -0.4328,E1 18.967,E2 515.9079} C_DIS
LIN {X 48.6445,Y -116.8759,Z 149,A -69.1177,B 18.8978,C -0.4298,E1 18.9633,E2 517.3404} C_DIS
LIN {X 45.5589,Y -118.1132,Z 149,A -70.5843,B 18.8978,C -0.4293,E1 18.9595,E2 518.8041} C_DIS
LIN {X 42.6546,Y -119.1928,Z 149,A -72.0941,B 18.8978,C -0.4234,E1 18.9555,E2 520.3276} C_DIS
LIN {X 38.4462,Y -120.6157,Z 149,A -74.0208,B 18.8978,C -0.4243,E1 18.9505,E2 522.2465} C_DIS
LIN {X 35.4779,Y -121.522,Z 149,A -75.5053,B 18.898,C -0.4198,E1 18.9464,E2 523.7414} C_DIS
LIN {X 30.9673,Y -122.749,Z 149,A -77.5132,B 18.898,C -0.4218,E1 18.9411,E2 525.7388} C_DIS
LIN {X 27.7296,Y -123.5215,Z 149,A -78.9738,B 18.898,C -0.4222,E1 18.9371,E2 527.1954} C_DIS
LIN {X 24.695,Y -124.1642,Z 149,A -80.3914,B 18.898,C -0.4206,E1 18.9332,E2 528.6156} C_DIS
LIN {X 21.871,Y -124.6922,Z 149,A -81.719,B 18.898,C -0.4186,E1 18.9296,E2 529.9473} C_DIS
LIN {X 18.5383,Y -125.2319,Z 149,A -83.2313,B 18.898,C -0.4182,E1 18.9254,E2 531.4589} C_DIS
LIN {X 15.6984,Y -125.6199,Z 149,A -84.5995,B 18.898,C -0.4147,E1 18.9216,E2 532.8362} C_DIS
LIN {X 12.6294,Y -125.9647,Z 149,A -85.9858,B 18.898,C -0.4145,E1 18.9177,E2 534.222} C_DIS
LIN {X 9.5489,Y -126.2349,Z 149,A -87.3257,B 18.898,C -0.4161,E1 18.914,E2 535.5559} C_DIS
LIN {X 6.2051,Y -126.4431,Z 149,A -88.7525,B 18.898,C -0.4189,E1 18.9101,E2 536.9734} C_DIS
LIN {X 3.085,Y -126.5584,Z 149,A -90.2192,B 18.898,C -0.4165,E1 18.9059,E2 538.447} C_DIS
LIN {X 0.9014,Y -126.5914,Z 149,A -90.934,B 18.8978,C -0.4265,E1 18.904,E2 539.1309} C_DIS
Enddeposition()
LIN {X 0.9412,Y -132.6149,Z 150,A -92.973,B 24.9685,C -1.2979,E1 25.0006,E2 539.5381} C_DIS
Startdeposition()
$VEL.CP = VEL_PRINT
LIN {X 3.4303,Y -132.5754,Z 150,A -91.2675,B 24.9668,C -1.3312,E1 25.0056,E2 537.7539} C_DIS
LIN {X 7.3919,Y -132.4154,Z 150,A -89.4469,B 24.9665,C -1.3376,E1 25.0107,E2 535.9188} C_DIS
LIN {X 11.3942,Y -132.1293,Z 150,A -87.8426,B 24.9668,C -1.3316,E1 25.0151,E2 534.3296} C_DIS
LIN {X 15.6229,Y -131.696,Z 150,A -86.0163,B 24.9668,C -1.3321,E1 25.0202,E2 532.5032} C_DIS
LIN {X 19.3031,Y -131.2082,Z 150,A -84.3037,B 24.9664,C -1.339,E1 25.025,E2 530.7758} C_DIS
LIN {X 23.1057,Y -130.5913,Z 150,A -82.7398,B 24.9666,C -1.335,E1 25.0292,E2 529.2231} C_DIS
LIN {X 26.5523,Y -129.9341,Z 150,A -81.2367,B 24.9666,C -1.3356,E1 25.0334,E2 527.7202} C_DIS
LIN {X 30.5866,Y -129.0449,Z 150,A -79.4769,B 24.9666,C -1.336,E1 25.0381,E2 525.962} C_DIS
LIN {X 33.9378,Y -128.2035,Z 150,A -77.9994,B 24.9666,C -1.3367,E1 25.0421,E2 524.485} C_DIS
LIN {X 37.0872,Y -127.328,Z 150,A -76.5691,B 24.9664,C -1.3393,E1 25.046,E2 523.051} C_DIS
LIN {X 40.3344,Y -126.3367,Z 150,A -75.1329,B 24.9664,C -1.3394,E1 25.0498,E2 521.6171} C_DIS
LIN {X 43.4525,Y -125.2985,Z 150,A -73.7321,B 24.9664,C -1.3402,E1 25.0535,E2 520.2172} C_DIS
LIN {X 46.4313,Y -124.2255,Z 150,A -72.4542,B 24.9665,C -1.3373,E1 25.0568,E2 518.949} C_DIS
LIN {X 49.3549,Y -123.0933,Z 150,A -70.9569,B 24.966,C -1.3469,E1 25.0608,E2 517.4322} C_DIS
LIN {X 52.4497,Y -121.8067,Z 150,A -69.4626,B 24.9658,C -1.3516,E1 25.0646,E2 515.9304} C_DIS
LIN {X 55.8814,Y -120.2711,Z 150,A -67.8933,B 24.9658,C -1.3512,E1 25.0686,E2 514.366} C_DIS
LIN {X 59.5849,Y -118.4815,Z 150,A -66.0528,B 24.9655,C -1.3576,E1 25.0733,E2 512.5153} C_DIS
LIN {X 63.1786,Y -116.6058,Z 150,A -64.262,B 24.9652,C -1.3628,E1 25.0777,E2 510.7173} C_DIS
LIN {X 67.1857,Y -114.3433,Z 150,A -62.3538,B 24.9652,C -1.3621,E1 25.0823,E2 508.8164} C_DIS
LIN {X 70.8852,Y -112.0875,Z 150,A -60.4537,B 24.965,C -1.3673,E1 25.0868,E2 506.9101} C_DIS
LIN {X 74.6489,Y -109.6175,Z 150,A -58.5077,B 24.9648,C -1.3713,E1 25.0913,E2 504.9612} C_DIS
LIN {X 78.1819,Y -107.1264,Z 150,A -56.6208,B 24.9645,C -1.3763,E1 25.0956,E2 503.0691} C_DIS
LIN {X 81.7589,Y -104.4214,Z 150,A -54.7189,B 24.9644,C -1.3786,E1 25.0998,E2 501.1686} C_DIS
LIN {X 85.3145,Y -101.5369,Z 150,A -52.7805,B 24.9643,C -1.381,E1 25.104,E2 499.2321} C_DIS
LIN {X 88.6751,Y -98.6159,Z 150,A -50.846,B 24.964,C -1.3861,E1 25.108,E2 497.2932} C_DIS
LIN {X 91.8472,Y -95.6686,Z 150,A -48.9769,B 24.9638,C -1.3906,E1 25.1118,E2 495.4212} C_DIS
LIN {X 94.816,Y -92.7268,Z 150,A -47.1947,B 24.9636,C -1.3938,E1 25.1154,E2 493.6389} C_DIS
LIN {X 97.8916,Y -89.4744,Z 150,A -45.2515,B 24.9633,C -1.3993,E1 25.1191,E2 491.6913} C_DIS
LIN {X 100.7664,Y -86.2243,Z 150,A -43.4037,B 24.9631,C -1.4028,E1 25.1224,E2 489.8436} C_DIS
LIN {X 103.4618,Y -82.9705,Z 150,A -41.5791,B 24.9629,C -1.4077,E1 25.1257,E2 488.0159} C_DIS
LIN {X 106.119,Y -79.5439,Z 150,A -39.6998,B 24.9626,C -1.4132,E1 25.1288,E2 486.1326} C_DIS
LIN {X 108.6388,Y -76.0662,Z 150,A -37.8476,B 24.9623,C -1.4183,E1 25.1318,E2 484.2774} C_DIS
LIN {X 111.1202,Y -72.3924,Z 150,A -36.0008,B 24.9623,C -1.42,E1 25.1347,E2 482.4357} C_DIS
LIN {X 113.3171,Y -68.9032,Z 150,A -34.1703,B 24.9618,C -1.428,E1 25.1374,E2 480.5958} C_DIS
LIN {X 115.6571,Y -64.8981,Z 150,A -32.3988,B 24.9622,C -1.421,E1 25.1398,E2 478.8498} C_DIS
LIN {X 118.4165,Y -59.7125,Z 150,A -29.6506,B 24.9611,C -1.4404,E1 25.1434,E2 476.0703} C_DIS
LIN {X 120.2604,Y -55.9046,Z 150,A -27.9631,B 24.9612,C -1.4383,E1 25.1454,E2 474.397} C_DIS
LIN {X 121.6174,Y -52.8877,Z 150,A -26.5362,B 24.961,C -1.4426,E1 25.147,E2 472.9677} C_DIS
LIN {X 122.9156,Y -49.7957,Z 150,A -25.1085,B 24.9608,C -1.446,E1 25.1485,E2 471.54} C_DIS
LIN {X 124.1963,Y -46.5093,Z 150,A -23.611,B 24.9606,C -1.4493,E1 25.15,E2 470.0429} C_DIS
LIN {X 125.3027,Y -43.4404,Z 150,A -22.2157,B 24.9604,C -1.453,E1 25.1513,E2 468.6466} C_DIS
LIN {X 126.3868,Y -40.1776,Z 150,A -20.7228,B 24.9602,C -1.4582,E1 25.1526,E2 467.15} C_DIS
LIN {X 127.5353,Y -36.3737,Z 150,A -18.9199,B 24.9596,C -1.4686,E1 25.1541,E2 465.3329} C_DIS
LIN {X 128.5319,Y -32.6714,Z 150,A -17.3695,B 24.9596,C -1.4681,E1 25.1551,E2 463.7927} C_DIS
LIN {X 129.3746,Y -29.1584,Z 150,A -15.7049,B 24.959,C -1.479,E1 25.1562,E2 462.112} C_DIS
LIN {X 130.228,Y -25.0712,Z 150,A -14.0237,B 24.959,C -1.4781,E1 25.1571,E2 460.4428} C_DIS
LIN {X 130.828,Y -21.7241,Z 150,A -12.5657,B 24.9588,C -1.4823,E1 25.1578,E2 458.9834} C_DIS
LIN {X 131.4401,Y -17.6515,Z 150,A -10.7581,B 24.9584,C -1.4898,E1 25.1585,E2 457.1688} C_DIS
LIN {X 131.875,Y -14.0328,Z 150,A -9.2041,B 24.9582,C -1.4938,E1 25.159,E2 455.6145} C_DIS
LIN {X 132.2621,Y -9.7298,Z 150,A -7.3541,B 24.9579,C -1.4991,E1 25.1594,E2 453.763} C_DIS
LIN {X 132.4999,Y -5.6516,Z 150,A -5.5663,B 24.9575,C -1.5062,E1 25.1597,E2 451.9691} C_DIS
LIN {X 132.6068,Y -1.87,Z 150,A -3.9169,B 24.9571,C -1.5125,E1 25.1597,E2 450.3148} C_DIS
LIN {X 132.5947,Y 2.5955,Z 150,A -1.9728,B 24.9567,C -1.5197,E1 25.1597,E2 448.3652} C_DIS
LIN {X 132.4539,Y 6.6257,Z 150,A -0.3484,B 24.9567,C -1.5188,E1 25.1595,E2 446.7525} C_DIS
LIN {X 132.1836,Y 10.7509,Z 150,A 1.456,B 24.9564,C -1.5257,E1 25.1592,E2 444.9425} C_DIS
LIN {X 131.8669,Y 14.1084,Z 150,A 2.8759,B 24.9562,C -1.5284,E1 25.1588,E2 443.5247} C_DIS
LIN {X 131.3965,Y 17.984,Z 150,A 4.6615,B 24.9556,C -1.5394,E1 25.1581,E2 441.7238} C_DIS
LIN {X 130.8425,Y 21.6373,Z 150,A 6.1153,B 24.9558,C -1.5367,E1 25.1575,E2 440.2849} C_DIS
LIN {X 130.2652,Y 24.8766,Z 150,A 7.5834,B 24.9553,C -1.5438,E1 25.1567,E2 438.8086} C_DIS
LIN {X 129.3642,Y 29.2043,Z 150,A 9.5073,B 24.9549,C -1.5507,E1 25.1556,E2 436.8797} C_DIS
LIN {X 128.0924,Y 34.3545,Z 150,A 11.7645,B 24.9546,C -1.556,E1 25.154,E2 434.623} C_DIS
LIN {X 126.8923,Y 38.5521,Z 150,A 13.5675,B 24.9546,C -1.5572,E1 25.1526,E2 432.8274} C_DIS
LIN {X 125.8601,Y 41.7982,Z 150,A 15.0346,B 24.9543,C -1.5615,E1 25.1513,E2 431.3585} C_DIS
LIN {X 124.7818,Y 44.9148,Z 150,A 16.4163,B 24.9542,C -1.5635,E1 25.1501,E2 429.9799} C_DIS
LIN {X 123.6483,Y 47.9471,Z 150,A 17.8301,B 24.9539,C -1.5685,E1 25.1487,E2 428.5621} C_DIS
LIN {X 122.4698,Y 50.8825,Z 150,A 19.1576,B 24.9538,C -1.5705,E1 25.1473,E2 427.2374} C_DIS
LIN {X 121.1522,Y 53.9445,Z 150,A 20.6257,B 24.9534,C -1.5763,E1 25.1456,E2 425.7637} C_DIS
LIN {X 119.7494,Y 56.9906,Z 150,A 22.0728,B 24.9532,C -1.5804,E1 25.1439,E2 424.3146} C_DIS
LIN {X 118.301,Y 59.9395,Z 150,A 23.5064,B 24.9529,C -1.5852,E1 25.1421,E2 422.8772} C_DIS
LIN {X 116.5772,Y 63.231,Z 150,A 25.2076,B 24.9523,C -1.595,E1 25.1398,E2 421.1619} C_DIS
LIN {X 114.2928,Y 67.2718,Z 150,A 27.145,B 24.9523,C -1.5968,E1 25.1371,E2 419.2303} C_DIS
LIN {X 111.9517,Y 71.1003,Z 150,A 29.0358,B 24.9521,C -1.5994,E1 25.1344,E2 417.343} C_DIS
LIN {X 109.621,Y 74.6437,Z 150,A 30.9406,B 24.9515,C -1.6082,E1 25.1314,E2 415.4269} C_DIS
LIN {X 107.0812,Y 78.2435,Z 150,A 32.8509,B 24.9512,C -1.6134,E1 25.1283,E2 413.5135} C_DIS
LIN {X 101.8921,Y 84.8909,Z 150,A 36.4438,B 24.9508,C -1.6196,E1 25.122,E2 409.9228} C_DIS
LIN {X 99.6177,Y 87.5487,Z 150,A 37.9861,B 24.9505,C -1.6248,E1 25.1192,E2 408.3751} C_DIS
LIN {X 96.5589,Y 90.9105,Z 150,A 39.8956,B 24.9505,C -1.6264,E1 25.1156,E2 406.4703} C_DIS
LIN {X 93.4156,Y 94.1373,Z 150,A 41.7744,B 24.9504,C -1.627,E1 25.1119,E2 404.598} C_DIS
LIN {X 87.4849,Y 99.6737,Z 150,A 45.3628,B 24.9497,C -1.6388,E1 25.1045,E2 400.9965} C_DIS
LIN {X 84.0818,Y 102.5602,Z 150,A 47.2458,B 24.9496,C -1.6401,E1 25.1004,E2 399.1175} C_DIS
LIN {X 80.6684,Y 105.266,Z 150,A 49.1043,B 24.9495,C -1.6424,E1 25.0964,E2 397.2604} C_DIS
LIN {X 77.1505,Y 107.8708,Z 150,A 50.9888,B 24.9493,C -1.6454,E1 25.0921,E2 395.3755} C_DIS
LIN {X 73.4177,Y 110.4455,Z 150,A 52.9551,B 24.949,C -1.6491,E1 25.0875,E2 393.4071} C_DIS
LIN {X 69.7016,Y 112.828,Z 150,A 54.8931,B 24.9487,C -1.6538,E1 25.083,E2 391.4643} C_DIS
LIN {X 65.8139,Y 115.1384,Z 150,A 56.804,B 24.9487,C -1.6544,E1 25.0784,E2 389.5577} C_DIS
LIN {X 62.111,Y 117.1763,Z 150,A 58.5987,B 24.9487,C -1.6553,E1 25.0739,E2 387.7661} C_DIS
LIN {X 58.8401,Y 118.8515,Z 150,A 60.1086,B 24.9487,C -1.6532,E1 25.0702,E2 386.265} C_DIS
LIN {X 55.7262,Y 120.3428,Z 150,A 61.591,B 24.9487,C -1.6546,E1 25.0665,E2 384.7834} C_DIS
LIN {X 52.157,Y 121.9333,Z 150,A 63.408,B 24.9482,C -1.6633,E1 25.0618,E2 382.95} C_DIS
LIN {X 48.6455,Y 123.3768,Z 150,A 65.0207,B 24.9482,C -1.6636,E1 25.0576,E2 381.3404} C_DIS
LIN {X 45.1121,Y 124.7107,Z 150,A 66.5376,B 24.9484,C -1.6591,E1 25.0537,E2 379.8373} C_DIS
LIN {X 41.8333,Y 125.8484,Z 150,A 68.0229,B 24.9484,C -1.6597,E1 25.0497,E2 378.3536} C_DIS
LIN {X 38.644,Y 126.8641,Z 150,A 69.5109,B 24.9482,C -1.663,E1 25.0458,E2 376.8603} C_DIS
LIN {X 35.9846,Y 127.6442,Z 150,A 70.9759,B 24.9472,C -1.6779,E1 25.0417,E2 375.3624} C_DIS
LIN {X 32.8863,Y 128.4773,Z 150,A 72.0894,B 24.9481,C -1.6645,E1 25.0388,E2 374.2824} C_DIS
LIN {X 29.1214,Y 129.3831,Z 150,A 73.8754,B 24.9477,C -1.6713,E1 25.0339,E2 372.4827} C_DIS
LIN {X 24.9875,Y 130.244,Z 150,A 75.5221,B 24.9482,C -1.6629,E1 25.0295,E2 370.8581} C_DIS
LIN {X 21.3239,Y 130.8948,Z 150,A 77.2642,B 24.9477,C -1.6705,E1 25.0246,E2 369.0999} C_DIS
LIN {X 17.5295,Y 131.4561,Z 150,A 78.8349,B 24.948,C -1.6664,E1 25.0203,E2 367.5401} C_DIS
LIN {X 14.1485,Y 131.8626,Z 150,A 80.3081,B 24.948,C -1.6668,E1 25.0162,E2 366.0671} C_DIS
LIN {X 10.3271,Y 132.2185,Z 150,A 82.0453,B 24.9477,C -1.671,E1 25.0114,E2 364.3208} C_DIS
LIN {X 6.609,Y 132.4547,Z 150,A 83.5979,B 24.9479,C -1.668,E1 25.0071,E2 362.7757} C_DIS
LIN {X 2.4595,Y 132.597,Z 150,A 85.3521,B 24.948,C -1.6658,E1 25.0022,E2 361.0272} C_DIS
LIN {X -0.8154,Y 132.6171,Z 150,A 86.8004,B 24.948,C -1.6673,E1 24.9981,E2 359.5756} C_DIS
LIN {X -4.9731,Y 132.5264,Z 150,A 88.5986,B 24.948,C -1.6668,E1 24.9931,E2 357.7782} C_DIS
LIN {X -8.882,Y 132.3237,Z 150,A 90.3965,B 24.9476,C -1.6716,E1 24.9881,E2 355.9684} C_DIS
LIN {X -12.7471,Y 132.0054,Z 150,A 91.9723,B 24.948,C -1.6657,E1 24.9837,E2 354.4058} C_DIS
LIN {X -16.6807,Y 131.5674,Z 150,A 94.1819,B 24.9465,C -1.6903,E1 24.9774,E2 352.1364} C_DIS
LIN {X -21.1152,Y 130.9296,Z 150,A 95.6836,B 24.9479,C -1.6667,E1 24.9734,E2 350.6893} C_DIS
LIN {X -24.693,Y 130.3004,Z 150,A 97.1705,B 24.9483,C -1.6613,E1 24.9694,E2 349.2136} C_DIS
LIN {X -27.954,Y 129.6397,Z 150,A 98.5636,B 24.9485,C -1.6578,E1 24.9656,E2 347.8272} C_DIS
LIN {X -31.3097,Y 128.8706,Z 150,A 100.138,B 24.9483,C -1.6608,E1 24.9613,E2 346.2436} C_DIS
LIN {X -35.4549,Y 127.7923,Z 150,A 101.9255,B 24.9486,C -1.6556,E1 24.9565,E2 344.4655} C_DIS
LIN {X -38.7147,Y 126.8425,Z 150,A 103.4279,B 24.9486,C -1.6558,E1 24.9525,E2 342.9602} C_DIS
LIN {X -41.9515,Y 125.809,Z 150,A 104.8708,B 24.9488,C -1.6527,E1 24.9486,E2 341.522} C_DIS
LIN {X -45.0132,Y 124.7463,Z 150,A 106.2585,B 24.949,C -1.6503,E1 24.945,E2 340.1373} C_DIS
LIN {X -47.922,Y 123.6581,Z 150,A 107.6357,B 24.949,C -1.6503,E1 24.9414,E2 338.7573} C_DIS
LIN {X -51.5203,Y 122.2034,Z 150,A 109.6117,B 24.9482,C -1.6629,E1 24.9362,E2 336.7469} C_DIS
LIN {X -56.4644,Y 120.0008,Z 150,A 111.7826,B 24.9489,C -1.6508,E1 24.9308,E2 334.5994} C_DIS
LIN {X -59.9103,Y 118.3158,Z 150,A 113.289,B 24.9496,C -1.6406,E1 24.927,E2 333.1133} C_DIS
LIN {X -63.12,Y 116.6376,Z 150,A 114.8623,B 24.9497,C -1.6382,E1 24.9232,E2 331.5411} C_DIS
LIN {X -67.6317,Y 114.0805,Z 150,A 117.5695,B 24.9485,C -1.6574,E1 24.9165,E2 328.7802} C_DIS
LIN {X -70.903,Y 112.0763,Z 150,A 118.8853,B 24.9498,C -1.6372,E1 24.9135,E2 327.5083} C_DIS
LIN {X -74.3098,Y 109.847,Z 150,A 120.6882,B 24.9498,C -1.6359,E1 24.9093,E2 325.7025} C_DIS
LIN {X -78.0416,Y 107.2282,Z 150,A 122.6491,B 24.9501,C -1.6314,E1 24.9049,E2 323.7456} C_DIS
LIN {X -81.5575,Y 104.5794,Z 150,A 124.5915,B 24.9503,C -1.6292,E1 24.9005,E2 321.8012} C_DIS
LIN {X -84.825,Y 101.9466,Z 150,A 126.3534,B 24.9507,C -1.6226,E1 24.8968,E2 320.0484} C_DIS
LIN {X -88.0605,Y 99.1652,Z 150,A 128.2368,B 24.9508,C -1.6203,E1 24.8928,E2 318.163} C_DIS
LIN {X -91.2011,Y 96.2846,Z 150,A 130.1017,B 24.951,C -1.6171,E1 24.889,E2 316.2983} C_DIS
LIN {X -93.5603,Y 93.9936,Z 150,A 131.8873,B 24.9501,C -1.6316,E1 24.8854,E2 314.4706} C_DIS
LIN {X -96.4102,Y 91.068,Z 150,A 133.275,B 24.9515,C -1.6085,E1 24.8828,E2 313.1317} C_DIS
LIN {X -99.3045,Y 87.903,Z 150,A 135.1514,B 24.9517,C -1.6049,E1 24.8793,E2 311.2556} C_DIS
Enddeposition()
END
